(* CODESYS project IndraLogic.project

Project tree, tasks and I/O mapping:
  IndraMotionMlc1 : IndraMotion MLC L45, Bosch Rexroth AG, order no. R911170828, version 13.12.1.0
    application Application
      libraries: ML_TechInterface, 13.12.0.0 (System); RIL_LoopControl, 13.12.0.0 (System); ML_TechMotion, 13.12.3.0 (System); ML_TechRegi, 13.12.0.0 (System); RIL_ModbusTCP, 13.12.0.0 (System); RMB_TechWinder, 13.12.0.0 (System)
      task PlcTask (cyclic, interval 10 ms, priority 2) calls MAIN
      task MotionTask (externalevent, external event EVENT_OP_MODE_MOTION_CYCLIC, priority 1) calls MOTION
      AdjustPreset/
        program AdjustPreset [ST]
        program WriteExpectWindow [LD]
      global variables UserConstGlobal
      trace Trace (task MotionTask): 
      program MAIN [ST]
      Expectation Window Managment/
        ML_RegiCtrlExpectWinType01/
          function block ML_RegiCtrlExpectWinType01 [ST]: actShutdown
          DataTypes/
            data type ML_REGICTRL_EXPECTWIN_TYPE01
        ML_WriteExpectWinPosEdgeType01/
          Datatypes/
            data type ML_WRITE_EXPECT_WIN_TYPE01
          function block ML_WriteExpectWinPosEdgeType01 [ST]
      global variables UserVarGlobal
      ModbusComDataType/
        data type REGISTER_DATA
      STATE_MACHINE/
        program Machine [ST]
        program Winder [ST]
      program FormatC [ST]
      data type SETUP_STATE
      global variables MlcVarGlobal
      global variables GVL_MODBUS
      REF_SPEED/
        program SetVmaSpeed [ST]
      data type UTIL_STATE
      MAIN_PGM/
        program GravureState [ST]
        program ModbusCom [ST]
      program InsetterControl [LD]
      FLEXO_PGM/
        program TouchProbe [ST]
        program ProbeSetup [ST]
      Symbols
      INFEED/
      program MOTION [ST]
      AxisInterface/
        program _Readme [ST]
        function block TE_AxisInterface [ST]: actRetriggerOpMode, actPMSpecialErrors, mClearError, actPhaseShift, actAngleOffset, mGetOpMode, mSetOpMode, actSetupMode, actSyncAccVel, actCopyAxisData_HMI, mInitExtension
        Visualizations/
          ImcInterface/
            visualisation ImcStatus
            visualisation ImcControl
            visualisation ImcInterface_Status_Control
          SystemOverview/
            visualisation System_Overview_header
            visualisation System_Overview
            visualisation System_Overview_All_Axis
          AxisModes/
            visualisation Velocity_mode
            visualisation Position_mode
            visualisation Profile_mode
            visualisation Axis_Overview
            visualisation Synchronization_mode
          Utilities/
            visualisation PLC_load
            visualisation AdjustPosition
            visualisation AdjustVelocity
        function block TE_AxisInitAllAxisType01 [ST]
        function Version_AxisInterface_13V600 [ST]
        Documentation/
          program Visualisierungen [ST]
          program Visualisations [ST]
        program TE_AxisInterfaceType01Prog [ST]: actInitWarmStart
        Type/
          Status/
            data type TE_AXIS_DIAGNOSIS
            data type TE_AXIS_ADMIN_STATUS
            data type TE_AXIS_DATA_STATUS
            data type TE_AXIS_VEL_STATUS
            data type TE_AXIS_STATUS_TYPE01
            data type TE_AXIS_SETUP_MODE_STATUS
            data type TE_AXIS_POS_STATUS
            data type TE_AXIS_SYNC_STATUS
          Control/
            data type TE_AXIS_SETUP_MODE
            data type TE_AXIS_SYNCHRONISATION
            data type TE_AXIS_VELOCITY
            data type TE_AXIS_CONTROL_TYPE01
            data type TE_AXIS_POSITIONING
            data type TE_AXIS_ADMINISTRATION
          data type TE_PLC_CYCLES_TIME
        global variables Global_Axis_Interface
      program AUTO_REGISTER [ST]
      Utilities/
        program AllAxisHealthy [ST]
        program AllAxisAB [ST]
        program UnSynchronizePullroll [ST]
        function block FB_writevar [ST]
        program SynchronizePullroll [ST]
        program UnSynchronizeFlexo [ST]
        program InitAxis [ST]
        program SynchronizeFlexo [ST]
      REWIND/
        program WinderProcess [ST]
      data type STATE
      program POU [ST]
    Sercos_III_Master : SercosIII Master, Rexroth, order no. 1, version 13.2.2.0
    Inline_I_O : Inline I/O, Bosch Rexroth AG, version 12.8.2.0
    Not_Used : Not Used, Bosch Rexroth AG, version 12.2.0.0
    Not_Used_1 : Not Used, Bosch Rexroth AG, version 12.2.0.0
    Onboard_I_O : Onboard I/O, Bosch Rexroth AG, version 13.6.2.0
        input  x1 : BOOL  // OnboardIn.1.1
        input  x2 : BOOL  // OnboardIn.2.1
        input  x3 : BOOL  // OnboardIn.1.4
        input  x4 : BOOL  // OnboardIn.2.4
        input  x5 : BOOL  // OnboardIn.1.1
        input  x6 : BOOL  // OnboardIn.2.1
        input  x7 : BOOL  // OnboardIn.1.4
        input  x8 : BOOL  // OnboardIn.2.4
        unmapped channels: OnboardIn, OnboardOut
  text list GlobalTextList
*)

// IndraMotionMlc1/Application/AxisInterface/Type/Control/TE_AXIS_SETUP_MODE
TYPE TE_AXIS_SETUP_MODE :
  STRUCT
	  (* Enable setup mode  | Freigabe Einrichtbetrieb
      - activates Power                        | - aktiviert Antriebsfreigabe *)
    Enable:          BOOL;
 
	  (* Jog +            | Tippen +
        - activates ModeVelocity with pos. Vel   | - aktiviert ModeVelocity mit pos. Vel *)
    JogPlus:         BOOL;
 
	  (* Jog -            | Tippen -
       - activates ModeVelocity with pos. Vel   | - aktiviert ModeVelocity mit neg. Vel *)
    JogMinus:        BOOL;

	  (* Homing
      - activates ModeHoming|SetAbsRef|ModesPosAbs | activiert ModeHoming|SetAbsRef|ModesPosAbs
        depending on axistype/-configuration       | abhängig vom Achstyp/-konfiguration       *) 
    Homing: BOOL;
	
    Vel:    REAL:= 10; (* jog/homing velocity  | Tipp-/Referenzfahrgeschwindigkeit *)
	
    Accel:  REAL:= 10; (* jog/homing ac/deceleration  | Tipp/Referenzfahr (brems)beschleunigung *)
  END_STRUCT
END_TYPE

// IndraMotionMlc1/Application/AxisInterface/Type/Control/TE_AXIS_SYNCHRONISATION
    (*************** - setpoint of synchronous motion ******************)
TYPE TE_AXIS_SYNCHRONISATION EXTENDS MB_AXIS_SYNCHRONISATION:
STRUCT

    (* Electronic gear input revolution
      - "ModeSyncPhase", "ModeSyncVel", "ModeSyncCam", "ModeSyncProfile", "ModeFlexProfile"
      - RatioNumerator for MC_GearIn, MB_GearInPos, MC_CamIn, MB_MotionProfile, ML_FlexProfile 
      Note: cyclic checked AND transmitted on change (EnableCyclicScanning = TRUE) 
      ------------------------------------------------------------------------------
      Elektronisches Getriebe, Eingangsumdrehungen
      - "ModeSyncPhase", "ModeSyncVel", "ModeSyncCam", "ModeSyncProfile", "ModeFlexProfile"
      - RatioNumerator fuer MC_GearIn, MB_GearInPos, MC_CamIn, MB_MotionProfile, ML_FlexProfile 
      Hinweis: wird permanent zyklisch verarbeitet (EnableCyclicScanning = TRUE) *)
    // InputRevolution: UINT:=1;

    (* Electronic gear output revolution
      - "ModeSyncPhase", "ModeSyncVel", "ModeSyncCam", "ModeSyncProfile", "ModeFlexProfile"
      - RatioDenominator for MC_GearIn, MB_GearInPos, MC_CamIn, MB_MotionProfile, ML_FlexProfile 
      Note: cyclic checked AND transmitted on change (EnableCyclicScanning = TRUE)
      ------------------------------------------------------------------------------
      Elektronisches Getriebe, Ausgangsumdrehungen
      - "ModeSyncPhase", "ModeSyncVel", "ModeSyncCam", "ModeSyncProfile", "ModeFlexProfile"
      - RatioDenominator fuer MC_GearIn, MB_GearInPos, MC_CamIn, MB_MotionProfile, ML_FlexProfile 
      Hinweis: wird permanent zyklisch verarbeitet (EnableCyclicScanning = TRUE) *)
    // OutputRevolution: UINT:=1;

    (* Master fine adjust
      - "ModeSyncPhase", "ModeSyncVel", "ModeSyncCam", "ModeSyncProfile", "ModeFlexProfile"
      - MasterFineadjust for MC_GearIn, MB_GearInPos, MC_CamIn, MB_MotionProfile, ML_FlexProfile
      Note: cyclic checked AND transmitted on change (EnableCyclicScanning = TRUE) 
      ------------------------------------------------------------------------------
      Getriebe-Feinabgleich
      - "ModeSyncPhase", "ModeSyncVel", "ModeSyncCam", "ModeSyncProfile", "ModeFlexProfile"
      - MasterFineadjust fuer MC_GearIn, MB_GearInPos, MC_CamIn, MB_MotionProfile, ML_FlexProfile
      Hinweis: wird permanent zyklisch verarbeitet (EnableCyclicScanning = TRUE) *)
    // FineAdjust:    REAL:=0.0;

    (* Cam Shaft Distance
      - start moving with "ModeSyncCam"
      - CamShaftDist for MC_CamIn
      Note: cyclic checked AND transmitted on change (EnableCyclicScanning = TRUE) 
      ------------------------------------------------------------------------------
      Kurvenscheibe, Hub
      - Freigabe mit "ModeSyncCam" 
      - CamShaftDist fuer MC_CamIn
      Hinweis: wird permanent zyklisch verarbeitet (EnableCyclicScanning = TRUE) *)
    // CamShaftDistance: REAL:=360.0;

    (* Phase offset between master and slave axis
      - "ModeSyncPhase", "ModeSyncCam", "ModeSyncProfile", "ModeFlexProfile" 
      - PhaseShift for MB_PhasingSlave
      Note: cyclic checked AND transmitted on change (EnableCyclicScanning = TRUE) 
      ------------------------------------------------------------------------------
      Winkelversatz (Lagesollwert additiv)
      - "ModeSyncPhase", "ModeSyncCam", "ModeSyncProfile", "ModeFlexProfile" 
      - PhaseShift fuer MB_PhasingSlave
      Hinweis: wird permanent zyklisch verarbeitet (EnableCyclicScanning = TRUE) *)
    // PhaseOffset:   REAL:=0.0; 

    (* Velocity for the phase offset
      - "ModeSyncPhase", "ModeSyncCam", "ModeSyncProfile", "ModeFlexProfile"
      - Velocity for MB_PhasingSlave 
      ------------------------------------------------------------------------------
      Aufsynchronisier-Geschwindigkeit
      - "ModeSyncPhase", "ModeSyncCam", "ModeSyncProfile", "ModeFlexProfile"
      - Velocity fuer MB_PhasingSlave *)
	// PhaseOffsetVel: REAL:=1.0;

    (* Acceleration for the phase offset
      - "ModeSyncPhase", "ModeSyncCam", "ModeSyncProfile", "ModeFlexProfile" 
      - PhaseShift for MB_PhasingSlave
      ------------------------------------------------------------------------------
      Aufsynchronisier-Beschleunigung
      - Freigabe mit "ModeSyncPhase", "ModeSyncCam" oder "ModeSyncProfile"
      - PhaseShift fuer MB_PhasingSlave *)
    // PhaseOffsetAcc: REAL:=100.0;

    (* Synchronisation direction
      - values 'SHORTEST_WAY'; 'CATCH_UP' (always forward); 'SLOW_DOWN' (see RIL_CommonTypes.lib)
      - start moving with "ModeSyncPhase", "ModeSyncCam" or "ModeSyncProfile"
      - SyncMode for MB_GearInPos, MC_CamIn, MB_MotionProfile 
      ------------------------------------------------------------------------------
      Aufsynchronisier-Richtung
      - Werte 'SHORTEST_WAY'; 'CATCH_UP' (positiv); 'SLOW_DOWN' (siehe RIL_CommonTypes.lib)
      - Freigabe mit "ModeSyncPhase", "ModeSyncCam" oder "ModeSyncProfile"
      - SyncMode fuer MB_GearInPos, MC_CamIn, MB_MotionProfile *)
    // SyncDirection: MC_SYNC_DIRECTION:= SHORTEST_WAY;

    (* Start mode of the synchronisation
      - values 'ABSOLUTE'; 'RELATIVE' (see RIL_CommonTypes.lib)
      - start moving with "ModeSyncPhase", "ModeSyncCam" or "ModeSyncProfile"
      - StartMode for MB_GearInPos, MC_CamIn, MB_MotionProfile 
      ------------------------------------------------------------------------------
      Aufsynchronisier-Mode
      - Werte: 'ABSOLUTE'; 'RELATIVE' (siehe RIL_CommonTypes.lib)
      - Freigabe mit "ModeSyncPhase", "ModeSyncCam" oder "ModeSyncProfile"
      - StartMode fuer MB_GearInPos, MC_CamIn, MB_MotionProfile *)
    // StartMode:     MC_START_MODE:= ABSOLUTE;

    (* Number of the selected cam table
      - values 'CAM_TABLE_1'; 'CAM_TABLE_2' ... 'CAM_TABLE_8' (see RIL_CommonTypes.lib)
      - start moving with "ModeSyncCam" 
      - CamTableID for MC_CamIn
      Note: cyclic checked AND transmitted on change (EnableCyclicScanning = TRUE)
      ------------------------------------------------------------------------------
      Nummer Stuetzpunkt-Tabelle
      - Werte: 'CAM_TABLE_1'; 'CAM_TABLE_2' ... 'CAM_TABLE_8' (siehe RIL_CommonTypes.lib)
      - Freigabe mit "ModeSyncCam" 
      - CamTableID fuer MC_CamIn
      Hinweis: wird permanent zyklisch verarbeitet (EnableCyclicScanning = TRUE) *)
    // CamTableID:    MC_CAM_ID:= CAM_TABLE_1;

    (* -> AXIS_REF of the master axis
      - "ModeSyncPhase", "ModeSyncVel", "ModeSyncCam", "ModeSyncProfile", "ModeFlexProfile"
      - Master for MC_GearIn, MB_GearInPos, MC_CamIn, MB_MotionProfile, ML_FlexProfile 
      Note: cyclic checked AND transmitted on change (EnableCyclicScanning = TRUE)
      ------------------------------------------------------------------------------
      -> AXIS_REF der Leitachse
      - "ModeSyncPhase", "ModeSyncVel", "ModeSyncCam", "ModeSyncProfile", "ModeFlexProfile"
      - Master fuer MC_GearIn, MB_GearInPos, MC_CamIn, MB_MotionProfile, ML_FlexProfile 
         Hinweis: wird permanent zyklisch verarbeitet (EnableCyclicScanning = TRUE) *)
    // Master:    AXIS_REF    := (AxisNo := NO_OBJECT, CntrlNo := LOCAL_CNTRL);


    (*************** Extensions for profile operation modes *******************)
    (************* Erweiterungen für die Profil Betriebsarten *****************)
    (* Extensions for the operating modes MotionProfile and FlexProfile
       ------------------------------------------------------------------------------
       Erweiterungen füt die Betriebsarten MotionProfile und FlexProfile *)
    // Profile:     ML_AXIS_PROFILE;
	
  (* add your extensions below here, keep the elements above
     Erweiterungen hier einfuegen, Elemente oberhalb nicht veraendern *)

  (* user extensions | Anwender Erweiterungen *)

  // angle offset begin of profile | Winkelverschiebung Tabellenanfang
	AngleOffset:   REAL:= 0;  
	
  // Values for MB_Phasing | Werte für MB_Phasing
  // Additive master position command value
	PhaseShift:    REAL:=0.0;    
	PhaseShiftVel: REAL:=10.0;   // Additive master position velocity  
	PhaseShiftAcc: REAL:=100.0;  // Additive master position acceleration
		
  // A-0-2790 Synchronisation velocity | Aufsynchronisiergeschw.
  SyncVelocity:     REAL := 10.0; 

	// A-0-2791 Synchron. acceleration | Aufsynchronisierbeschleunigung
  SyncAcceleration: REAL := 10.0; 

END_STRUCT
END_TYPE

// IndraMotionMlc1/Application/AxisInterface/Type/Status/TE_AXIS_DIAGNOSIS
    (********** Diagnosis outputs - from motion control to logic control *****************)
    (********** Diagnose-Ausgaenge - Motion Control zur Logic Control    *****************)
TYPE TE_AXIS_DIAGNOSIS EXTENDS MB_AXIS_DIAGNOSIS:

STRUCT

  (* add your extensions below here |  Erweiterungen hier einfuegen*)

  (* user extensions | Anwender Erweiterungen *)


END_STRUCT

END_TYPE

// IndraMotionMlc1/Application/AxisInterface/Type/Control/TE_AXIS_VELOCITY
    (*************** - setpoints of velocity mode                    ************)
    (*************** - Sollwerte Geschwindigkeitsregelung (Freilauf) ************)
TYPE TE_AXIS_VELOCITY EXTENDS MB_AXIS_VELOCITY:
STRUCT

    (* Value of the maximum velocity (Unit: [u/s])
      - start moving with "ModeVel" (MC_MoveVelocity)
      Note: cyclic checked AND transmitted on change (EnableCyclicScanning = TRUE) 
      -----------------------------------------------------------------------------
      Geschwindigkeits-Sollwert, (Einheit: [u/s]) 
      - Freigabe mit "ModeVel" (MC_MoveVelocity)
      Hinweis: wird permanent zyklisch verarbeitet (EnableCyclicScanning = TRUE) *)
    // Velocity:        REAL:=0.0;

    (* Value of the acceleration and deceleration [u/s2] (always positive)
      - start moving with "ModeVel" (MC_MoveVelocity)
      -----------------------------------------------------------------------------
      Beschleunigung, (Einheit: [u/s2]) (immer positiv eingeben)            
      - Freigabe mit "ModeVel" (MC_MoveVelocity) *)
    // Acceleration:    REAL:=10.0;

    (* Value of the deceleration [u/s2] (always positive)
      - start moving with "ModeVel" (MC_MoveVelocity) 
      -----------------------------------------------------------------------------
      Verzoegerung, (Einheit: [u/s2]) (immer positiv eingeben)
      - Freigabe mit "ModeVel" (MC_MoveVelocity) *)
    // Deceleration:    REAL:=10.0;
	
(* add your extensions below here, keep the elements above
   Erweiterungen hier einfuegen, Elemente oberhalb nicht veraendern *)

(* user extensions | Anwender Erweiterungen *)

END_STRUCT
END_TYPE

// IndraMotionMlc1/Application/SETUP_STATE
TYPE SETUP_STATE :
(
	MECH_ACTIVE,MECH_UNSYNC,MECH_FORMAT_CH_P2,WRITE_NEW_GEARING,MECH_FORMAT_CH_P4,MECH_RESYNC,MECH_ERROR
);
END_TYPE

// IndraMotionMlc1/Application/AxisInterface/Type/Status/TE_AXIS_ADMIN_STATUS
    (********** Administrative outputs - from motion control to logic control *****************)
    (********** Administrative Ausgaenge - Motion Control zur Logic Control   *****************)
TYPE TE_AXIS_ADMIN_STATUS EXTENDS MB_AXIS_ADMIN_STATUS:

STRUCT
  (* add your extensions below here |  Erweiterungen hier einfuegen*)

  (* User extensions | Anwender Erweiterungen *)

 
END_STRUCT

END_TYPE

// IndraMotionMlc1/Application/AxisInterface/Type/Status/TE_AXIS_DATA_STATUS
TYPE TE_AXIS_DATA_STATUS :
STRUCT
	                  dwMotionProfileStatusBits_i     :DWORD;      (* A-0-2931 -RD- Motion profile status word *)
                      FlexProfil_Sync                 :BOOL;       (* A-0-3010.08 -RD- FlexProfile is in synchronisation *)
                      FlexProfil_Active               :BOOL;       (* A-0-3010.09 -RD- FlexProfile is active *)
                      FlexProfil_WaitForSwitching     :BOOL;       (* A-0-3010.10 -RD- FlexProfile is waiting for switching position *)
                      FlexProfil_Set0_Checked         :BOOL;       (* A-0-3010.16 -RD- FlexProfile Set0 is checked *)
                      FlexProfil_Set0_Ok              :BOOL;       (* A-0-3010.17 -RD- FlexProfile Set0 is ok *)
                      FlexProfil_Set1_Checked         :BOOL;       (* A-0-3010.18 -RD- FlexProfile Set0 is checked *)
                      FlexProfil_Set1_Ok              :BOOL;       (* A-0-3010.19 -RD- FlexProfile Set0 is ok *)
                      FlexProfil_Set2_Checked         :BOOL;       (* A-0-3010.20 -RD- FlexProfile Set0 is checked *)
                      FlexProfil_Set2_Ok              :BOOL;       (* A-0-3010.21 -RD- FlexProfile Set0 is ok *)
                      FlexProfil_Set3_Checked         :BOOL;       (* A-0-3010.22 -RD- FlexProfile Set0 is checked *)
                      FlexProfil_Set3_Ok              :BOOL;       (* A-0-3010.23 -RD- FlexProfile Set0 is ok *)
                      FlexProfil_EvtSet0_Checked      :BOOL;       (* A-0-3010.24 -RD- FlexProfile Event Set0 is checked *)
                      FlexProfil_EvtSet0_Ok           :BOOL;       (* A-0-3010.25 -RD- FlexProfile Event Set0 is ok *)
                      FlexProfil_EvtSet1_Checked      :BOOL;       (* A-0-3010.26 -RD- FlexProfile Event Set0 is checked *)
                      FlexProfil_EvtSet1_Ok           :BOOL;       (* A-0-3010.27 -RD- FlexProfile Event Set0 is ok *)
                      FlexProfil_EvtSet2_Checked      :BOOL;       (* A-0-3010.28 -RD- FlexProfile Event Set0 is checked *)
                      FlexProfil_EvtSet2_Ok           :BOOL;       (* A-0-3010.29 -RD- FlexProfile Event Set0 is ok *)
                      FlexProfil_EvtSet3_Checked      :BOOL;       (* A-0-3010.30 -RD- FlexProfile Event Set0 is checked *)
                      FlexProfil_EvtSet3_Ok           :BOOL;       (* A-0-3010.31 -RD- FlexProfile Event Set0 is ok *)
                      dwFlexProfileEventStatusBits_i  :DWORD;      (* A-0-3012 -RD- Condition status variable, FlexProfile *)

                      Axis_CamTab_0                   :BOOL;       (* A-0-0021.00 -RD- Cam shaft table BOOL 0 *)                
                      Axis_CamTab_1                   :BOOL;       (* A-0-0021.01 -RD- Cam shaft table BOOL 1 *)
                      Axis_CamTab_2                   :BOOL;       (* A-0-0021.02 -RD- Cam shaft table BOOL 2 (reserved) *)
                      Axis_CamSwitching               :BOOL;       (* A-0-0021.03 -RD- Status cam shaft distance switching *)
                      Axis_InVelocity                 :BOOL;       (* A-0-0021.04 -RD- Axis cmd velocity == actual velocity *)
                      Axis_Standstill                 :BOOL;       (* A-0-0021.05 -RD- Axis velocity <= A-0-0222 (standstill) *)
                      Axis_InPosition                 :BOOL;       (* A-0-0021.06 -RD- Axis cmd position == actual position *)
                      Axis_InSynchron                 :BOOL;       (* A-0-0021.07 -RD- Axis is in synchronisation *)
                      Axis_Warning                    :BOOL;       (* A-0-0021.08 -RD- Axis reports warning *)
                      Axis_Error                      :BOOL;       (* A-0-0021.09 -RD- Axis reports error *)
                      Axis_Homed                      :BOOL;       (* A-0-0021.10 -RD- Axis is relative / in homing *)
                      Axis_InTorque                   :BOOL;       (* A-0-0021.11 -RD- Axis cmd torque / force == actual torque *)
                      Axis_OperationMode              :BOOL;       (* A-0-0021.12 -RD- Axis is in operation mode (P4) *)
                      Axis_Inbb                       :BOOL;       (* A-0-0021.13 -RD- Axis is ready for power to the amplifier (bb) *)
                      Axis_InAb                       :BOOL;       (* A-0-0021.14 -RD- Axis is ready for power to the engine (Ab) *)
                      Axis_Power                      :BOOL;       (* A-0-0021.15 -RD- Axis has power on (AH_AF) *)
                      Axis_CmdActive                  :BOOL;       (* A-0-0021.16 -RD- Command active *)
                      Axis_ErrInProgress              :BOOL;       (* A-0-0021.17 -RD- Error reaction in progress *)
                      Axis_CyclicPosChannelOpen       :BOOL;       (* A-0-0021.18 -RD- Cyclic Position Channel is open for Axis *)          
                      Axis_InMasterPhaseOffset        :BOOL;       (* A-0-0021.19 -RD- Master Phase offset achieved *)
                      Axis_CyclicTrqChannelOpen       :BOOL;       (* A-0-0021.20 -RD- Cyclic Position Channel is open for Axis *)          
                      Axis_CyclicVelChannelOpen       :BOOL;       (* A-0-0021.21 -RD- Cyclic Position Channel is open for Axis *)          
                      Axis_CyclicAnaChannelOpen       :BOOL;       (* A-0-0021.22 -RD- Cyclic Position Channel is open for Axis *)          
                      ErrorStop                       :BOOL;       (* A-0-0022.00 -RD- Axis is in "ErrorStop" *)
                      Stopping                        :BOOL;       (* A-0-0022.01 -RD- Axis is in "Stopping" *)
                      Homing                          :BOOL;       (* A-0-0022.02 -RD- Command homing is active *)
                      PowerOn                         :BOOL;       (* A-0-0022.03 -RD- Axis got power *)
                      DiscreteMotion                  :BOOL;       (* A-0-0022.04 -RD- Axis is in "Discrete Motion" *)
                      ContinuousMotion                :BOOL;       (* A-0-0022.05 -RD- Axis is in "Continuous Motion" *)
                      SynchronizedMotion              :BOOL;       (* A-0-0022.06 -RD- Axis is in "Synchronized Motion" *)
                      Standstill                      :BOOL;       (* A-0-0022.07 -RD- Axis is stopped *)
                      CoordinatedMotion               :BOOL;       (* A-0-0022.08 -RD- Axis is in "CoordinatedMotion" *)
                      ControlledMotion                :BOOL;       (* A-0-0022.09 -RD- Axis is in "ControlledMotion" *)  
                      dwAxisCondition_i               :DWORD;      (* A-0-0024 -RD- Axis condition *)
                      rActualPosition_i               :REAL;       (* A-0-0100 -RD- Actual position *)
                      rActualVelocity_i               :REAL;       (* A-0-0102 -RD- Actual velocity *)
                      rActualTorqueForce_i            :REAL;       (* A-0-0110 -RD- Actual torque/force *)
                                                                                 
                    
                      wUserActualDataBitA_i           :WORD;      (* A-0-0562 -RD- User defined actual data BOOL number A, Type: WORD *)
                      wUserActualDataBitB_i           :WORD;      (* A-0-0565 -RD- User defined actual data BOOL number B, Type: WORD *)
                      wUserActualDataBitC_i           :WORD;      (* A-0-0568 -RD- User defined actual data BOOL number C, Type: WORD *)
                      wUserActualDataBitD_i           :WORD;      (* A-0-0571 -RD- User defined actual data BOOL number D, Type: WORD *)
                    
                      dwUserActualDataA_i             :SM_TYPES;  (* A-0-0521 -RD- Container user defined actual data A *)
                      dwUserActualDataB_i             :SM_TYPES;  (* A-0-0523 -RD- Container user defined actual data B *)
                      dwUserActualDataC_i             :SM_TYPES;  (* A-0-0525 -RD- Container user defined actual data C *)
                      dwUserActualDataD_i             :SM_TYPES;  (* A-0-0527 -RD- Container user defined actual data D *)
                      dwUserActualDataE_i             :SM_TYPES;  (* A-0-0529 -RD- Container user defined actual data E *)
                      dwUserActualDataF_i             :SM_TYPES;  (* A-0-0531 -RD- Container user defined actual data F *)
END_STRUCT
END_TYPE

// IndraMotionMlc1/Application/Expectation Window Managment/ML_WriteExpectWinPosEdgeType01/Datatypes/ML_WRITE_EXPECT_WIN_TYPE01
TYPE ML_WRITE_EXPECT_WIN_TYPE01 :
(
	STATE_IDLE,
	STATE_CHECK_VALIDITY,
	STATE_CALC_WINDOWS,
	STATE_WRITE_START_POS,
	STATE_WRITE_END_POS,
	STATE_ERROR,
	STATE_DONE,
	STATE_SHUTDOWN,
	STATE_RESET_PARAM_INST,
	STATE_DUMMY

);
END_TYPE

// IndraMotionMlc1/Application/AxisInterface/Type/Status/TE_AXIS_VEL_STATUS
    (********* Outputs of the following axis - from motion control to logic control **********)
    (********* Achs-Ausgaenge - Motion Control zur Logic Control                    **********)
TYPE TE_AXIS_VEL_STATUS  EXTENDS MB_AXIS_VEL_STATUS:
STRUCT
	(* -> outputs of the adjusting functionality for the velocity
      -> Ausgaenge fuer Tippbetrieb der Geschwindigkeit *)
    //Adjust: MB_AXIS_ADJUST_STATUS;
 
(* add your extensions below here, keep the elements above
   Erweiterungen hier einfuegen, Elemente oberhalb nicht veraendern *)

(* user extensions | Anwender Erweiterungen *)

END_STRUCT

END_TYPE

// IndraMotionMlc1/Application/AxisInterface/Type/Status/TE_AXIS_STATUS_TYPE01
    (********* Outputs of the following axis - from motion control to logic control **********)
TYPE TE_AXIS_STATUS_TYPE01:
  STRUCT
    (********* Outputs of the following axis - from motion control to logic control **********)

    PtrAxisData:  POINTER TO ML_AXISDATA_SM;
     (* Pointer to AxisData of this axis | Zeiger auf AxisData dieser Achse
      - Type .PtrAxisData^. for the intellisense menu | Eingabe .PtrAxisData^. fuer Auswahlmenue*)

    Admin:   TE_AXIS_ADMIN_STATUS; (* status of the axis | Achs-Status *)

    Diag:    TE_AXIS_DIAGNOSIS; (* axis diagnosis information, error, warning....
      Diagnose Informationen der Achse, Fehler, Warnung.... *)

    PosMode: TE_AXIS_POS_STATUS; (* Status operating mode positioning (absolute, rel. and add.)
      Statusmeldungen Positionierbetrieb (absolut, relativ und additiv) *)

    VelMode: TE_AXIS_VEL_STATUS; (* Status operating mode velocity control
      Statusmeldungen Geschwindigkeitsregelung (Freilauf) *)

    SyncMode: TE_AXIS_SYNC_STATUS; (* Status operating mode synchronisation (phase, vel, and cam)
      Statusmeldungen Synchronbetriebsarten (Winkelsync., Geschwindigkeitssync. und Kurvensch.)*)

    (* add your extensions below here, keep the elements above
       Erweiterungen hier einfuegen, Elemente oberhalb nicht veraendern *)
    (* user extensions | Anwender Erweiterungen *)
		(* Jog/Homing functionality | Tipp/Einrichtfunktionen *)
    SetupMode:  TE_AXIS_SETUP_MODE_STATUS;

    // AxisData for HMI (without data type "BIT")
	  AxisData_HMI:	TE_AXIS_DATA_STATUS;
	
  END_STRUCT
END_TYPE

// IndraMotionMlc1/Application/AxisInterface/Type/Status/TE_AXIS_SETUP_MODE_STATUS
TYPE TE_AXIS_SETUP_MODE_STATUS :
  STRUCT
	  (* Acknowledge setup mode  | Bestätigung Einrichtbetrieb
      - removed when _OpMode is oerwritten | - wird weggenommen, wenn _OpMode überschrieben wird *)
    EnableAck:   BOOL;
 
	  (* Acknowledge Homing 
      - ModeHoming|SetAbsRef|ModesPosAbs | ModeHoming|SetAbsRef|ModesPosAbs
        finished                         | abgeschlossen                    *) 
    HomingAck: 		BOOL;
	
  END_STRUCT
END_TYPE

// IndraMotionMlc1/Application/UTIL_STATE
TYPE UTIL_STATE :
(COMMAND,WAIT,DONE);
END_TYPE

// IndraMotionMlc1/Application/AxisInterface/Type/Control/TE_AXIS_CONTROL_TYPE01
TYPE TE_AXIS_CONTROL_TYPE01:

STRUCT
    Admin:      TE_AXIS_ADMINISTRATION; (* Administration of the axis | Verwaltung der Achse *)

    PosMode:    TE_AXIS_POSITIONING; (* operating mode positioning (absolute, rel. and additive)
      Positionierbetrieb (absolut, relativ und additiv) *)

    VelMode:    TE_AXIS_VELOCITY; (* operating mode velocity control | Geschwindigkeitsregelung *)

    SyncMode:   TE_AXIS_SYNCHRONISATION; (* operating mode synchronisation (phase, vel, and cam)
      Synchronbetriebsarten (Winkelsync., Geschwindigkeitssync. und Kurvenscheibe) *)

    (* add your extensions below here, keep the elements above
       Erweiterungen hier einfuegen, Elemente oberhalb nicht veraendern *)

    (* user extensions | Anwender Erweiterungen *)
    
	  // Jog/Homing functionality | Tipp/Einrichtfunktionen 
    SetupMode:  TE_AXIS_SETUP_MODE; 
	
END_STRUCT

END_TYPE

// IndraMotionMlc1/Application/ModbusComDataType/REGISTER_DATA
TYPE REGISTER_DATA :
STRUCT
	arWord:    ARRAY[0..20]OF WORD;     (* 1000 WORDS (%MB0000 - %MB999 ) *)
    (*arInt:     ARRAY[0..999]OF INT;      (* 1000 WORDS (%MB1000 - %MB1999) *)
	arUint:    ARRAY[0..999]OF UINT;     (* 1000 WORDS (%MB2000 - %MB2999) *)
	arDint:    ARRAY[0..499]OF DINT;     (* 1000 WORDS (%MB3000 - %MB3999) *)
	arUdint:   ARRAY[0..499]OF UDINT;    (* 1000 WORDS (%MB4000 - %MB4999) *)
	arReal:    ARRAY[0..499]OF REAL;     (* 1000 WORDS (%MB5000 - %MB5999) *)
	arString:  ARRAY[0..99]OF STRING(19);(* 1000 WORDS (%MB6000 - %MB6999) *)
	(* String(19): because 19 byte string + 1 byte end sign *)
	(* together 7000 WORDS *)*)
END_STRUCT
END_TYPE

// IndraMotionMlc1/Application/AxisInterface/Type/Status/TE_AXIS_POS_STATUS
    (********* Outputs of the following axis - from motion control to logic control **********)
    (********* Achs-Ausgaenge - Motion Control zur Logic Control                    **********)
TYPE TE_AXIS_POS_STATUS EXTENDS MB_AXIS_POS_STATUS:
STRUCT

	(* -> outputs of the adjusting functionality for the position
      -> Ausgaenge fuer Tippbetrieb der Position *)
    //Adjust: MB_AXIS_ADJUST_STATUS;
 
(* add your extensions below here, keep the elements above
   Erweiterungen hier einfuegen, Elemente oberhalb nicht veraendern *)

(* user extensions | Anwender Erweiterungen *)

END_STRUCT

END_TYPE

// IndraMotionMlc1/Application/AxisInterface/Type/Control/TE_AXIS_POSITIONING
    (*************** - setpoints of positioning mode ******************)
    (*************** - Positions-Sollwerte           ******************)
TYPE TE_AXIS_POSITIONING EXTENDS MB_AXIS_POSITIONING:
STRUCT

    (* position for an absolute move (in technical unit[u]) (negative or positive)
      - start moving with "ModePosAbs" (MC_MoveAbsolute)
      Note: cyclic checked AND transmitted on change (EnableCyclicScanning = TRUE) 
      ------------------------------------------------------------------------------
      Zielposition, absolut (Einheit: [u]) (negativ oder positiv)
      - Freigabe mit "ModePosAbs" (MC_MoveAbsolute)
      Hinweis: wird permanent zyklisch verarbeitet (EnableCyclicScanning = TRUE) *)
    // Position:        REAL;

    (* distance for a relative or additive move (in technical unit[u]) (negative or positive)
      - start moving with "ModePosRel" or "ModePosAdd" (MC_MoveRelative, MC_MoveAdditive) 
      Note: cyclic checked AND transmitted on change (EnableCyclicScanning = TRUE) 
      ------------------------------------------------------------------------------
      Relativer / additiver Sollwert (Einheit: [u]) (negativ oder positiv )
      - Freigabe mit "ModePosRel" oder "ModePosAdd" (MC_MoveRelative, MC_MoveAdditive) 
      Hinweis: wird permanent zyklisch verarbeitet (EnableCyclicScanning = TRUE) *)
     // Distance:        REAL;

    (* maximum velocity (always positive) (not necessarily reached) [u/s]
      - start moving with "ModePosAbs" or "ModePosRel" or "ModePosAdd" 
        (MC_MoveAbsolute, MC_MoveRelative, MC_MoveAdditive) 
      Note: cyclic checked AND transmitted on change (EnableCyclicScanning = TRUE) 
      ------------------------------------------------------------------------------
      Positioniergeschwindigkeit , (Einheit: [u/s]) (positiv eingeben)
      - Freigabe mit "ModePosAbs" oder "ModePosRel" oder "ModePosAdd" 
        (MC_MoveAbsolute, MC_MoveRelative, MC_MoveAdditive) 
      Hinweis: wird permanent zyklisch verarbeitet (EnableCyclicScanning = TRUE) *)
    // Velocity:        REAL:=10.0;

    (* Value of the acceleration (always positive) (increasing energy of the motor) [u/s2]
      - start moving with "ModePosAbs" or "ModePosRel" or "ModePosAdd" 
        (MC_MoveAbsolute, MC_MoveRelative, MC_MoveAdditive) 
      ------------------------------------------------------------------------------
      Beschleunigung (Einheit: [u/s2]) (nur positive Werte)             
      - Freigabe mit "ModePosAbs" oder "ModePosRel" oder "ModePosAdd" 
        (MC_MoveAbsolute, MC_MoveRelative, MC_MoveAdditive) *)
    // Acceleration:    REAL:=10.0;

    (* Value of the deceleration (always positive) (decreasing energy of the motor) [u/s2]
      - start moving with ModePosAbs or ModePosRel or ModePosAdd 
        (MC_MoveAbsolute, MC_MoveRelative, MC_MoveAdditive) 
      ------------------------------------------------------------------------------
      Verzoegerung, (Einheit: [u/s2]) (nur positive Werte)            
      - Freigabe mit "ModePosAbs" oder "ModePosRel" oder "ModePosAdd" 
        (MC_MoveAbsolute, MC_MoveRelative, MC_MoveAdditive) *)
    // Deceleration:    REAL:=10.0;
	
(* add your extensions below here, keep the elements above
   Erweiterungen hier einfuegen, Elemente oberhalb nicht veraendern *)

(* user extensions | Anwender Erweiterungen *)

END_STRUCT
END_TYPE

// IndraMotionMlc1/Application/AxisInterface/Type/Control/TE_AXIS_ADMINISTRATION
TYPE TE_AXIS_ADMINISTRATION EXTENDS MB_AXIS_ADMINISTRATION:
STRUCT
  (* add your extensions below here |  Erweiterungen hier einfuegen*)

  (* user extensions | Anwender Erweiterungen *)
  
  // Restart the same OpMode again, e.g. MoveRelative with same distance
  RetriggerOpMode: BOOL;	

END_STRUCT
END_TYPE

// IndraMotionMlc1/Application/AxisInterface/Type/Status/TE_AXIS_SYNC_STATUS
    (********* Outputs of the following axis - from motion control to logic control **********)
    (********* Achs-Ausgaenge - Motion Control zur Logic Control                    **********)
TYPE TE_AXIS_SYNC_STATUS EXTENDS MB_AXIS_SYNC_STATUS:
STRUCT
    // CamActiveID:      MC_CAM_ID; (* - ID of the active CamTable | - Nr. aktive Stuetzpunkt-Tab.*)

	(* - Number of the active motion profile set 0 or 1
      - Nummer des aktiven Satzes 0 oder 1 des Bewegungsprofils *)
    // ProfileActiveSet: UINT:= 0;  

	(* - Change of PhaseOffset is finished
      - Verstellung des PhaseOffset ist abgeschlossen  *)
    // PhasingSlaveDone: BOOL := FALSE; 

	(* adjusting | vertippen
      arAxisCntrl[].SyncMode.FineAdjust *)
    //AdjFineAdjust:       MB_AXIS_ADJUST_STATUS; 

	(* adjusting | vertippen
      arAxisCntrl[].SyncMode.CamShaftDistance *)
    //AdjCamShaftDistance: MB_AXIS_ADJUST_STATUS; 

	(* adjusting | vertippen
      arAxisCntrl[].SyncMode.PhaseOffset *)
    //AdjPhaseOffset:      MB_AXIS_ADJUST_STATUS;
	
  (* add your extensions below here, keep the elements above
     Erweiterungen hier einfuegen, Elemente oberhalb nicht veraendern *)

  (* user extensions | Anwender Erweiterungen *)
	// angle offset begin of profile | Winkelverschiebung Tabellenanfang 
  // transmission done | Übertragung abgeschlossen  
	AngleOffsetDone:   BOOL:= FALSE;   

  // Synchronisation velocity | Aufsynchronisiergeschw.
  // transmission done | Übertragung abgeschlossen  
  SyncVelocityDone:  BOOL:= FALSE;     

	// Synchron. acceleration | Aufsynchronisierbeschleunigung
  // transmission done | Übertragung abgeschlossen 
  SyncAccelerationDone: BOOL:= FALSE;  
	
  // Change of PhaseShift is finished | Verstellung des PhaseShift ist abgeschlossen 
  PhasingMasterDone: BOOL:=FALSE;
 
END_STRUCT

END_TYPE

// IndraMotionMlc1/Application/STATE

	
TYPE STATE :
(ERROR_CHECK,SETUP_PREPARE,SETUP_WAIT,SETUP_P2,SETUP_WRITEGEAR,SETUP_WRITEGEAR_WAIT,SETUP_P4,INIT_SYNC,INIT_VERIFY,
HOLD,RUN_PREPARE,RUN_DELAY,RUN,JOG_PREPARE,JOG_DELAY,JOG,JOG_WAIT,ERROR);


END_TYPE

// IndraMotionMlc1/Application/AxisInterface/Type/TE_PLC_CYCLES_TIME
TYPE TE_PLC_CYCLES_TIME :
STRUCT

     udiMinimumTime  : UDINT  := 1000000;
     udiActualTime   : UDINT  := 0;
     udiMaximumTime  : UDINT  := 0;

END_STRUCT
END_TYPE

// IndraMotionMlc1/Application/Expectation Window Managment/ML_RegiCtrlExpectWinType01/DataTypes/ML_REGICTRL_EXPECTWIN_TYPE01
TYPE ML_REGICTRL_EXPECTWIN_TYPE01 :
(
	
	STATE_IDLE,
	STATE_STORAGE_MODE_OFF,
	STATE_WAIT_REGI_IN_OPERATION,
	STATE_RESET_FB_INST,
	STATE_WAIT_REGI_SETPOINT_LOCK,
	STATE_RUN,
	STATE_SHUTDOWN,
	STATE_ERROR,
	STATE_DUMMY
);
END_TYPE

// IndraMotionMlc1/Application/UserConstGlobal
VAR_GLOBAL CONSTANT
  // define all possible axis, set to maximum axis index to preserve ressources 
  // set to a maximum of 32 for the L45 and 16? for the L25
  uiMAX_AXIS_INDEX:   UINT    := INT_TO_UINT(MB_MAX_AXIS_NUMBER);

  uiPRINT_AXIS_INDEX: UINT :=2;
END_VAR

// IndraMotionMlc1/Application/UserVarGlobal
VAR_GLOBAL 
  // Axis interface: command structure: define as RETAIN, to keep the values 
  // Note: on the L40.2 control, the RETAIN memory is slower then normal VAR, so define 
  //       this structure only as RETAIN when necessary 
  //  arAxisCtrl_gb: ARRAY [1..MAX_AXIS_NUM] OF MB_AXIS_CONTROL;
	
  // Axis interface: command structure 
  arAxisCtrl_gb: ARRAY [1..uiMAX_AXIS_INDEX] OF TE_AXIS_CONTROL_TYPE01;
	rExpectWindowPosEdgeStart_gb: REAL;
	rExpectWindowPosEdgeEnd_gb: REAL;
	rSetPointWindows_gb: REAL;
	Probe1Infeed: TOUCHPROBE_REF := (TouchProbeNo := TOUCHPROBE_DRIVE_1, CntrlNo := LOCAL_CNTRL);
END_VAR

VAR_GLOBAL
//----------------------------------- Machine status variables ----------------------------	

  // Axis interface: status structure 
  arAxisStatus_gb: ARRAY [1..uiMAX_AXIS_INDEX] OF TE_AXIS_STATUS_TYPE01;

  bRemoteOn_gb  : BOOL := TRUE;  // TRUE: Internal IL visu is active 
                                 // FALSE: PlcProg is active

								 	(*DEFINITION DU TOUCHPROB*)
tpDrv1: TOUCHPROBE_REF := (TouchProbeNo := TOUCHPROBE_DRIVE_1, CntrlNo := LOCAL_CNTRL);
  
END_VAR

// IndraMotionMlc1/Application/MlcVarGlobal
(* Automatically generated code by XLC/MLC. *)
(* Please don't edit, the code will be overwritten. For usercode use UserVarGlobal! *)
{attribute 'linkalways'}
VAR_GLOBAL CONSTANT

(*Real axis "Drive1" with axis number 1*)
Drive1: AXIS_REF :=(CntrlNo:=LOCAL_CNTRL,AxisNo:=AXIS_1);

(*Real axis "Drive2" with axis number 2*)
Drive2: AXIS_REF :=(CntrlNo:=LOCAL_CNTRL,AxisNo:=AXIS_2);

(*Real axis "Drive20" with axis number 20*)
Drive20: AXIS_REF :=(CntrlNo:=LOCAL_CNTRL,AxisNo:=AXIS_20);

(*Virtual axis "VMA_FT1" with axis number 30*)
VMA_FT1: AXIS_REF :=(CntrlNo:=LOCAL_CNTRL,AxisNo:=AXIS_30);


(*Probe 001*)
TouchProbe001: TOUCHPROBE_REF :=(CntrlNo:=LOCAL_CNTRL,TouchProbeNo:=TOUCHPROBE_1);

(*Probe 002*)
TouchProbe002: TOUCHPROBE_REF :=(CntrlNo:=LOCAL_CNTRL,TouchProbeNo:=TOUCHPROBE_2);

(*Probe 003*)
TouchProbe003: TOUCHPROBE_REF :=(CntrlNo:=LOCAL_CNTRL,TouchProbeNo:=TOUCHPROBE_3);

(*Probe 004*)
TouchProbe004: TOUCHPROBE_REF :=(CntrlNo:=LOCAL_CNTRL,TouchProbeNo:=TOUCHPROBE_4);

(*Probe 005*)
TouchProbe005: TOUCHPROBE_REF :=(CntrlNo:=LOCAL_CNTRL,TouchProbeNo:=TOUCHPROBE_5);

(*Probe 006*)
TouchProbe006: TOUCHPROBE_REF :=(CntrlNo:=LOCAL_CNTRL,TouchProbeNo:=TOUCHPROBE_6);

(*Probe 007*)
TouchProbe007: TOUCHPROBE_REF :=(CntrlNo:=LOCAL_CNTRL,TouchProbeNo:=TOUCHPROBE_7);

(*Probe 008*)
TouchProbe008: TOUCHPROBE_REF :=(CntrlNo:=LOCAL_CNTRL,TouchProbeNo:=TOUCHPROBE_8);

(*Probe 009*)
TouchProbe009: TOUCHPROBE_REF :=(CntrlNo:=LOCAL_CNTRL,TouchProbeNo:=TOUCHPROBE_9);

(*Probe 010*)
TouchProbe010: TOUCHPROBE_REF :=(CntrlNo:=LOCAL_CNTRL,TouchProbeNo:=TOUCHPROBE_10);

(*Probe 011*)
TouchProbe011: TOUCHPROBE_REF :=(CntrlNo:=LOCAL_CNTRL,TouchProbeNo:=TOUCHPROBE_11);

(*Probe 012*)
TouchProbe012: TOUCHPROBE_REF :=(CntrlNo:=LOCAL_CNTRL,TouchProbeNo:=TOUCHPROBE_12);

(*Probe 013*)
TouchProbe013: TOUCHPROBE_REF :=(CntrlNo:=LOCAL_CNTRL,TouchProbeNo:=TOUCHPROBE_13);

(*Probe 014*)
TouchProbe014: TOUCHPROBE_REF :=(CntrlNo:=LOCAL_CNTRL,TouchProbeNo:=TOUCHPROBE_14);

(*Probe 015*)
TouchProbe015: TOUCHPROBE_REF :=(CntrlNo:=LOCAL_CNTRL,TouchProbeNo:=TOUCHPROBE_15);

(*Probe 016*)
TouchProbe016: TOUCHPROBE_REF :=(CntrlNo:=LOCAL_CNTRL,TouchProbeNo:=TOUCHPROBE_16);

(*Probe 017*)
TouchProbe017: TOUCHPROBE_REF :=(CntrlNo:=LOCAL_CNTRL,TouchProbeNo:=TOUCHPROBE_17);

(*Probe 018*)
TouchProbe018: TOUCHPROBE_REF :=(CntrlNo:=LOCAL_CNTRL,TouchProbeNo:=TOUCHPROBE_18);

(*Probe 019*)
TouchProbe019: TOUCHPROBE_REF :=(CntrlNo:=LOCAL_CNTRL,TouchProbeNo:=TOUCHPROBE_19);

(*Probe 020*)
TouchProbe020: TOUCHPROBE_REF :=(CntrlNo:=LOCAL_CNTRL,TouchProbeNo:=TOUCHPROBE_20);

(*Probe 021*)
TouchProbe021: TOUCHPROBE_REF :=(CntrlNo:=LOCAL_CNTRL,TouchProbeNo:=TOUCHPROBE_21);

(*Probe 022*)
TouchProbe022: TOUCHPROBE_REF :=(CntrlNo:=LOCAL_CNTRL,TouchProbeNo:=TOUCHPROBE_22);

(*Probe 023*)
TouchProbe023: TOUCHPROBE_REF :=(CntrlNo:=LOCAL_CNTRL,TouchProbeNo:=TOUCHPROBE_23);

(*Probe 024*)
TouchProbe024: TOUCHPROBE_REF :=(CntrlNo:=LOCAL_CNTRL,TouchProbeNo:=TOUCHPROBE_24);

(*Probe 025*)
TouchProbe025: TOUCHPROBE_REF :=(CntrlNo:=LOCAL_CNTRL,TouchProbeNo:=TOUCHPROBE_25);

(*Probe 026*)
TouchProbe026: TOUCHPROBE_REF :=(CntrlNo:=LOCAL_CNTRL,TouchProbeNo:=TOUCHPROBE_26);

(*Probe 027*)
TouchProbe027: TOUCHPROBE_REF :=(CntrlNo:=LOCAL_CNTRL,TouchProbeNo:=TOUCHPROBE_27);

(*Probe 028*)
TouchProbe028: TOUCHPROBE_REF :=(CntrlNo:=LOCAL_CNTRL,TouchProbeNo:=TOUCHPROBE_28);

(*Probe 029*)
TouchProbe029: TOUCHPROBE_REF :=(CntrlNo:=LOCAL_CNTRL,TouchProbeNo:=TOUCHPROBE_29);

(*Probe 030*)
TouchProbe030: TOUCHPROBE_REF :=(CntrlNo:=LOCAL_CNTRL,TouchProbeNo:=TOUCHPROBE_30);

(*Probe 031*)
TouchProbe031: TOUCHPROBE_REF :=(CntrlNo:=LOCAL_CNTRL,TouchProbeNo:=TOUCHPROBE_31);

(*Probe 032*)
TouchProbe032: TOUCHPROBE_REF :=(CntrlNo:=LOCAL_CNTRL,TouchProbeNo:=TOUCHPROBE_32);

(*Probe 033*)
TouchProbe033: TOUCHPROBE_REF :=(CntrlNo:=LOCAL_CNTRL,TouchProbeNo:=TOUCHPROBE_33);

(*Probe 034*)
TouchProbe034: TOUCHPROBE_REF :=(CntrlNo:=LOCAL_CNTRL,TouchProbeNo:=TOUCHPROBE_34);

(*Probe 035*)
TouchProbe035: TOUCHPROBE_REF :=(CntrlNo:=LOCAL_CNTRL,TouchProbeNo:=TOUCHPROBE_35);

(*Probe 036*)
TouchProbe036: TOUCHPROBE_REF :=(CntrlNo:=LOCAL_CNTRL,TouchProbeNo:=TOUCHPROBE_36);

(*Probe 037*)
TouchProbe037: TOUCHPROBE_REF :=(CntrlNo:=LOCAL_CNTRL,TouchProbeNo:=TOUCHPROBE_37);

(*Probe 038*)
TouchProbe038: TOUCHPROBE_REF :=(CntrlNo:=LOCAL_CNTRL,TouchProbeNo:=TOUCHPROBE_38);

(*Probe 039*)
TouchProbe039: TOUCHPROBE_REF :=(CntrlNo:=LOCAL_CNTRL,TouchProbeNo:=TOUCHPROBE_39);

(*Probe 040*)
TouchProbe040: TOUCHPROBE_REF :=(CntrlNo:=LOCAL_CNTRL,TouchProbeNo:=TOUCHPROBE_40);

(*Probe 041*)
TouchProbe041: TOUCHPROBE_REF :=(CntrlNo:=LOCAL_CNTRL,TouchProbeNo:=TOUCHPROBE_41);

(*Probe 042*)
TouchProbe042: TOUCHPROBE_REF :=(CntrlNo:=LOCAL_CNTRL,TouchProbeNo:=TOUCHPROBE_42);

(*Probe 043*)
TouchProbe043: TOUCHPROBE_REF :=(CntrlNo:=LOCAL_CNTRL,TouchProbeNo:=TOUCHPROBE_43);

(*Probe 044*)
TouchProbe044: TOUCHPROBE_REF :=(CntrlNo:=LOCAL_CNTRL,TouchProbeNo:=TOUCHPROBE_44);

(*Probe 045*)
TouchProbe045: TOUCHPROBE_REF :=(CntrlNo:=LOCAL_CNTRL,TouchProbeNo:=TOUCHPROBE_45);

(*Probe 046*)
TouchProbe046: TOUCHPROBE_REF :=(CntrlNo:=LOCAL_CNTRL,TouchProbeNo:=TOUCHPROBE_46);

(*Probe 047*)
TouchProbe047: TOUCHPROBE_REF :=(CntrlNo:=LOCAL_CNTRL,TouchProbeNo:=TOUCHPROBE_47);

(*Probe 048*)
TouchProbe048: TOUCHPROBE_REF :=(CntrlNo:=LOCAL_CNTRL,TouchProbeNo:=TOUCHPROBE_48);

(*Probe 049*)
TouchProbe049: TOUCHPROBE_REF :=(CntrlNo:=LOCAL_CNTRL,TouchProbeNo:=TOUCHPROBE_49);

(*Probe 050*)
TouchProbe050: TOUCHPROBE_REF :=(CntrlNo:=LOCAL_CNTRL,TouchProbeNo:=TOUCHPROBE_50);

(*Probe 051*)
TouchProbe051: TOUCHPROBE_REF :=(CntrlNo:=LOCAL_CNTRL,TouchProbeNo:=TOUCHPROBE_51);

(*Probe 052*)
TouchProbe052: TOUCHPROBE_REF :=(CntrlNo:=LOCAL_CNTRL,TouchProbeNo:=TOUCHPROBE_52);

(*Probe 053*)
TouchProbe053: TOUCHPROBE_REF :=(CntrlNo:=LOCAL_CNTRL,TouchProbeNo:=TOUCHPROBE_53);

(*Probe 054*)
TouchProbe054: TOUCHPROBE_REF :=(CntrlNo:=LOCAL_CNTRL,TouchProbeNo:=TOUCHPROBE_54);

(*Probe 055*)
TouchProbe055: TOUCHPROBE_REF :=(CntrlNo:=LOCAL_CNTRL,TouchProbeNo:=TOUCHPROBE_55);

(*Probe 056*)
TouchProbe056: TOUCHPROBE_REF :=(CntrlNo:=LOCAL_CNTRL,TouchProbeNo:=TOUCHPROBE_56);

(*Probe 057*)
TouchProbe057: TOUCHPROBE_REF :=(CntrlNo:=LOCAL_CNTRL,TouchProbeNo:=TOUCHPROBE_57);

(*Probe 058*)
TouchProbe058: TOUCHPROBE_REF :=(CntrlNo:=LOCAL_CNTRL,TouchProbeNo:=TOUCHPROBE_58);

(*Probe 059*)
TouchProbe059: TOUCHPROBE_REF :=(CntrlNo:=LOCAL_CNTRL,TouchProbeNo:=TOUCHPROBE_59);

(*Probe 060*)
TouchProbe060: TOUCHPROBE_REF :=(CntrlNo:=LOCAL_CNTRL,TouchProbeNo:=TOUCHPROBE_60);

(*Probe 061*)
TouchProbe061: TOUCHPROBE_REF :=(CntrlNo:=LOCAL_CNTRL,TouchProbeNo:=TOUCHPROBE_61);

(*Probe 062*)
TouchProbe062: TOUCHPROBE_REF :=(CntrlNo:=LOCAL_CNTRL,TouchProbeNo:=TOUCHPROBE_62);

(*Probe 063*)
TouchProbe063: TOUCHPROBE_REF :=(CntrlNo:=LOCAL_CNTRL,TouchProbeNo:=TOUCHPROBE_63);

(*Probe 064*)
TouchProbe064: TOUCHPROBE_REF :=(CntrlNo:=LOCAL_CNTRL,TouchProbeNo:=TOUCHPROBE_64);

(*Probe 065*)
TouchProbe065: TOUCHPROBE_REF :=(CntrlNo:=LOCAL_CNTRL,TouchProbeNo:=TOUCHPROBE_65);

(*Probe 066*)
TouchProbe066: TOUCHPROBE_REF :=(CntrlNo:=LOCAL_CNTRL,TouchProbeNo:=TOUCHPROBE_66);

(*Probe 067*)
TouchProbe067: TOUCHPROBE_REF :=(CntrlNo:=LOCAL_CNTRL,TouchProbeNo:=TOUCHPROBE_67);

(*Probe 068*)
TouchProbe068: TOUCHPROBE_REF :=(CntrlNo:=LOCAL_CNTRL,TouchProbeNo:=TOUCHPROBE_68);

(*Probe 069*)
TouchProbe069: TOUCHPROBE_REF :=(CntrlNo:=LOCAL_CNTRL,TouchProbeNo:=TOUCHPROBE_69);

(*Probe 070*)
TouchProbe070: TOUCHPROBE_REF :=(CntrlNo:=LOCAL_CNTRL,TouchProbeNo:=TOUCHPROBE_70);

(*Probe 071*)
TouchProbe071: TOUCHPROBE_REF :=(CntrlNo:=LOCAL_CNTRL,TouchProbeNo:=TOUCHPROBE_71);

(*Probe 072*)
TouchProbe072: TOUCHPROBE_REF :=(CntrlNo:=LOCAL_CNTRL,TouchProbeNo:=TOUCHPROBE_72);

(*Probe 073*)
TouchProbe073: TOUCHPROBE_REF :=(CntrlNo:=LOCAL_CNTRL,TouchProbeNo:=TOUCHPROBE_73);

(*Probe 074*)
TouchProbe074: TOUCHPROBE_REF :=(CntrlNo:=LOCAL_CNTRL,TouchProbeNo:=TOUCHPROBE_74);

(*Probe 075*)
TouchProbe075: TOUCHPROBE_REF :=(CntrlNo:=LOCAL_CNTRL,TouchProbeNo:=TOUCHPROBE_75);

(*Probe 076*)
TouchProbe076: TOUCHPROBE_REF :=(CntrlNo:=LOCAL_CNTRL,TouchProbeNo:=TOUCHPROBE_76);

(*Probe 077*)
TouchProbe077: TOUCHPROBE_REF :=(CntrlNo:=LOCAL_CNTRL,TouchProbeNo:=TOUCHPROBE_77);

(*Probe 078*)
TouchProbe078: TOUCHPROBE_REF :=(CntrlNo:=LOCAL_CNTRL,TouchProbeNo:=TOUCHPROBE_78);

(*Probe 079*)
TouchProbe079: TOUCHPROBE_REF :=(CntrlNo:=LOCAL_CNTRL,TouchProbeNo:=TOUCHPROBE_79);

(*Probe 080*)
TouchProbe080: TOUCHPROBE_REF :=(CntrlNo:=LOCAL_CNTRL,TouchProbeNo:=TOUCHPROBE_80);

(*Probe 081*)
TouchProbe081: TOUCHPROBE_REF :=(CntrlNo:=LOCAL_CNTRL,TouchProbeNo:=TOUCHPROBE_81);

(*Probe 082*)
TouchProbe082: TOUCHPROBE_REF :=(CntrlNo:=LOCAL_CNTRL,TouchProbeNo:=TOUCHPROBE_82);

(*Probe 083*)
TouchProbe083: TOUCHPROBE_REF :=(CntrlNo:=LOCAL_CNTRL,TouchProbeNo:=TOUCHPROBE_83);

(*Probe 084*)
TouchProbe084: TOUCHPROBE_REF :=(CntrlNo:=LOCAL_CNTRL,TouchProbeNo:=TOUCHPROBE_84);

(*Probe 085*)
TouchProbe085: TOUCHPROBE_REF :=(CntrlNo:=LOCAL_CNTRL,TouchProbeNo:=TOUCHPROBE_85);

(*Probe 086*)
TouchProbe086: TOUCHPROBE_REF :=(CntrlNo:=LOCAL_CNTRL,TouchProbeNo:=TOUCHPROBE_86);

(*Probe 087*)
TouchProbe087: TOUCHPROBE_REF :=(CntrlNo:=LOCAL_CNTRL,TouchProbeNo:=TOUCHPROBE_87);

(*Probe 088*)
TouchProbe088: TOUCHPROBE_REF :=(CntrlNo:=LOCAL_CNTRL,TouchProbeNo:=TOUCHPROBE_88);

(*Probe 089*)
TouchProbe089: TOUCHPROBE_REF :=(CntrlNo:=LOCAL_CNTRL,TouchProbeNo:=TOUCHPROBE_89);

(*Probe 090*)
TouchProbe090: TOUCHPROBE_REF :=(CntrlNo:=LOCAL_CNTRL,TouchProbeNo:=TOUCHPROBE_90);

(*Probe 091*)
TouchProbe091: TOUCHPROBE_REF :=(CntrlNo:=LOCAL_CNTRL,TouchProbeNo:=TOUCHPROBE_91);

(*Probe 092*)
TouchProbe092: TOUCHPROBE_REF :=(CntrlNo:=LOCAL_CNTRL,TouchProbeNo:=TOUCHPROBE_92);

(*Probe 093*)
TouchProbe093: TOUCHPROBE_REF :=(CntrlNo:=LOCAL_CNTRL,TouchProbeNo:=TOUCHPROBE_93);

(*Probe 094*)
TouchProbe094: TOUCHPROBE_REF :=(CntrlNo:=LOCAL_CNTRL,TouchProbeNo:=TOUCHPROBE_94);

(*Probe 095*)
TouchProbe095: TOUCHPROBE_REF :=(CntrlNo:=LOCAL_CNTRL,TouchProbeNo:=TOUCHPROBE_95);

(*Probe 096*)
TouchProbe096: TOUCHPROBE_REF :=(CntrlNo:=LOCAL_CNTRL,TouchProbeNo:=TOUCHPROBE_96);

(*Probe 097*)
TouchProbe097: TOUCHPROBE_REF :=(CntrlNo:=LOCAL_CNTRL,TouchProbeNo:=TOUCHPROBE_97);

(*Probe 098*)
TouchProbe098: TOUCHPROBE_REF :=(CntrlNo:=LOCAL_CNTRL,TouchProbeNo:=TOUCHPROBE_98);

(*Probe 099*)
TouchProbe099: TOUCHPROBE_REF :=(CntrlNo:=LOCAL_CNTRL,TouchProbeNo:=TOUCHPROBE_99);

(*Probe 100*)
TouchProbe100: TOUCHPROBE_REF :=(CntrlNo:=LOCAL_CNTRL,TouchProbeNo:=TOUCHPROBE_100);

END_VAR

// IndraMotionMlc1/Application/GVL_MODBUS
VAR_GLOBAL
	

	//RegisterData:          REGISTER_DATA;              (* Holding Register data area for FC3, FC6, FC16 and FC23        *)
	bGratuve_Tens_Inc_ETH_i	:BOOL;
	bGratuve_Tens_Dec_ETH_i	:BOOL;
	bGravure_Reg_Adv_ETH_q	:BOOL;
	bGravure_Reg_Ret_ETH_q	:BOOL;
	bGravureOn_ETH_q		:BOOL;
	
	bRegAdvance_ETH_i		:BOOL;
	bRegRetard_ETH_i		:BOOL;
	bGravure_Jog_Adv_HMI_i	:BOOL;
	bGravure_Jog_Ret_HMI_i	:BOOL;
	
	bInfeedOn_ETH_q			:BOOL;
	bInfeedManual_ETH_q		:BOOL;
	bInfeed_Inc_Tens_HMI_i	:BOOL;
	bInfeed_Dec_Tens_HMI_i	:BOOL;
	
	uiGearingRatio_HMI_q	:BOOL;
	
	bGravure_StatusError_HMI_q		:BOOL;
	bGravure_StatusSynch_HMI_q		:BOOL;
	bGravure_StatusSlowRot_HMI_q	:BOOL;
	bGravure_StatusDisabled_HMI_q	:BOOL;
	
	bInfeed_StatusError_HMI_q		:BOOL;
	bInfeed_StatusSynch_HMI_q		:BOOL;
	bInfeed_StatusSlowRot_HMI_q		:BOOL;
	bInfeed_StatusDisabled_HMI_q	:BOOL;
	
	bGravure_ResetDrive_HMI_i:BOOL;
	bInfeed_ResetDrive_HMI_i:BOOL;
	bRewindPID_Out_i:BOOL;
	bGravureSlowRot_ETH_i:BOOL;
	
	
		bGravureFB:BOOL:= TRUE;
		bGravureRegiOn_HMI_i:	BOOL;
		bInfeedRegiOn_HMI_i:	BOOL;
		bGravureNipActive_i:	BOOL;
		bPauseRegiOn_HMI_i: BOOL;
		bSetPtLckRegiCtrl_HMI_i: BOOL;
		bSetPtLckRegiCtrlAck_HMI_q: BOOL;
		bTouchProbeInOp_HMI_q:BOOL;
		uiDetectedPosEdge_gb:UINT;
		rCurrentValue_HMI_q:REAL;
		rRegiCtrlSetPoint: REAL;
		rDeviation_gb:REAL;
	
		rDeviationMil_gb:REAL;
		rSetPointWindowsMil_gb:REAL;
		
		
		
	dwDeviation_gb:DWORD;
	dwDeviation_low_gb:DWORD;
	dwDeviation_high_gb:DWORD;


	dwRegiCtrlSetPoint_gb:DWORD;
	dwRegiCtrlSetPoint_low_gb:DWORD;
	dwRegiCtrlSetPoint_high_gb:DWORD;
	dwLoadcellTension_gb:DWORD;
	
	dwRegAdjustLow_gb:DWORD;
	dwRegAdjustHigh_gb:DWORD;
	dwRegAdjust_gb:DWORD;
	
	arDrive: ARRAY[1..2] OF AXIS_REF;
	arProbe: ARRAY[1..2] OF TOUCHPROBE_REF;
END_VAR

// IndraMotionMlc1/Application/AxisInterface/Global_Axis_Interface
{attribute 'linkalways'}
VAR_GLOBAL
    (* Axis number for the visualization screens *)
    VisuAxisNo : INT := 1;
END_VAR

// IndraMotionMlc1/Application/MAIN
PROGRAM MAIN
VAR
	
ii:UINT;
bBogus:BOOL;
uiState1:UTIL_STATE;
uiState2:UTIL_STATE;
bRun_HMI_i:BOOL;
bJog_HMI_i:BOOL;
bStop_HMI_i:BOOL;
bReset_HMI_i:BOOL;
bOkToRun_i:BOOL:=TRUE;
bOkToJog_i:BOOL:=TRUE;
bFault_i:BOOL;
bInterlock_i:BOOL:=TRUE;
bSetup_HMI_i:BOOL;
newSTATE:STATE;
bSetupDone_i:BOOL;

	arFlexoAxis:	ARRAY[1..20] OF AXIS_REF;
	arPullrollAxis: ARRAY[1..20] OF AXIS_REF;
	arWindingAxis:	ARRAY[1..20] OF AXIS_REF;
	
	index:UINT;
		
	arFlexoPointer: POINTER TO ARRAY[1..20] OF AXIS_REF;
	test:AXIS_REF;
	uiAxisTotNumNew: UINT;
	
	
	bUnsync:BOOL;
	bSync:BOOL;
	binit:BOOL:=FALSE;	
	bAllAxisAB:BOOL;
	bAllFlexoSync:BOOL;
	bAllFlexoUnsync: BOOL;
	
	fbRunButton: R_TRIG;
	fbSetupButton: R_TRIG;
	
	rRepeat_i	:REAL	:= 1.0;
	iFormat_i	:INT := 4800;	//8 inches format
	rRunSpd		:REAL:= 100.0;
	rJogSpd		:REAL:= 10.0;
	bWriteExec: BOOL;
	
	bRewIntrlock:BOOL;
END_VAR


VAR CONSTANT
	uiNUM_FLEXO		: UINT:=2;
	uiNUM_PULLROLL	: UINT:=0;
	uiNUM_WINDER	: UINT:=1;
	iTeethConstant	: INT :=8;
END_VAR

IF TE_AxisInterfaceType01Prog.InitDone=FALSE THEN
	RETURN;
END_IF

//AXIS DEFINITION
arFlexoAxis[1] := arAxisCtrl_gb[Drive1.AxisNo].Admin.Axis;
arFlexoAxis[2] := arAxisCtrl_gb[Drive2.AxisNo].Admin.Axis;
//Winders
arWindingAxis[1]:= arAxisCtrl_gb[Drive20.AxisNo].Admin.Axis;

IF NOT binit THEN InitAxis(arAxisPointer:=ADR(arFlexoAxis) , uiNUM_FLEXO_F:= uiNUM_FLEXO);
				  InitAxis(arAxisPointer:=ADR(arWindingAxis) , uiNUM_FLEXO_F:= uiNUM_WINDER);

ELSE	//______    INIT IS OVER       ______!!!!!!!



bReset_HMI_i;
//THIS FUNCTION IS THE CORE OF THE MACHINE POSSIBLE STATES
Winder(
	arAxisPointer:= ADR(arWindingAxis), 
	uiNUM_FLEXO_F:= uiNUM_WINDER, 
	MACHINE_STATE_i:= newSTATE, 
	iGearValue:= 1, 
	bRewIntrlock=> bRewIntrlock);


Machine(
	arAxisPointer_M	:=ADR(arFlexoAxis),
	uiNUM_FLEXO_M	:=uiNUM_FLEXO,
	bRun_i			:=	bRun_HMI_i , 
	bJog_i			:=	bJog_HMI_i , 
	bStop_i			:=	bStop_HMI_i , 
	okToRun			:=	bOkToRun_i , 
	okToJog			:=	bOkToJog_i , 
	bFault			:=	bFault_i, 
	bIntrlock		:=	bInterlock_i, 
	bSetup_i		:=	 bSetup_HMI_i,
	bWriteExec		:=  bWriteExec, 
	CURRENT_STATE_OUT=> newSTATE );	

rRepeat_i:=INT_TO_REAL(iFormat_i/iTeethConstant)/ 100.0;

//THIS FUNCTION SETS SPEED ACCORDING TO THE FORMAT 
SetVmaSpeed(
	arAxisPointer:=ADR(arFlexoAxis) , 
	uiNUM_FLEXO_F:=uiNUM_FLEXO , 
	rFormat:=rRepeat_i , 
	rRunSpeedDemandFPM:=rRunSpd , 
	rJogSpeedDemandFPM:= rJogSpd, 
	uiState:=newSTATE , 
	);
//SET FORMAT
//THIS FUNCTION SETS MECHANICAL GEAR DEPENDING ON THE PLATE CYLINDER USED
//IT ALSO ADJUSTS THE SYNC_REVOLUTION TO COMPENSATES THE ADJUSTMENT OF VMA SPEED
FormatC(
	arAxisPointer:= ADR(arFlexoAxis), 
	uiNUM_FLEXO_F:= uiNUM_FLEXO , 
	MACHINE_STATE_i:= newSTATE , 
	iGearValue:=     iFormat_i , 
	bExecute:= bWriteExec , 
	bSetupDone_i=> );	

//GravureState();
//InfeedState();
ModbusCom();
//POU();

END_IF
binit:= TRUE;

END_PROGRAM

// IndraMotionMlc1/Application/AxisInterface/TE_AxisInterfaceType01Prog
PROGRAM TE_AxisInterfaceType01Prog
(*#############################################################################################
  #############################################################################################  

   General Header   
  ---------------------------------------------------------------------------------------------  
   Shortdescription       : Cyclic execution of the Axis-Interface (POS, VEL and SYNC mode)
   Version                : see Version_GAT_compact_11V200 
   Name                   : DCC/EAM3 (KG)
   Date                   : see Version_GAT_compact_11V200
   Company                : see Version_GAT_compact_11V200
   Target                 : see Version_GAT_compact_11V200
   Functional description : This program executes cyclic the axis interface FB for all axes.
                            The execution time of the axis interface FB is measured.
   Handling specials      : The global arrays of the axis-interface must be named arAxisCtrl[]
                            and arAxisStatus[]
  ---------------------------------------------------------------------------------------------  
    
   Additional Header   
  ---------------------------------------------------------------------------------------------  
  #############################################################################################  
  #############################################################################################*)
(*
                                     ******************
                                     *   DISCLAIMER   *
                                     ******************
   It is acknowledged that with regard to these software programs and program modules free of
   charge, Bosch Rexroth's usually practised, in-house test and release procedures have not 
   been accomplished. These software programs and program modules free of charge serve only as
   an example for possible applications.  They are intended as a help in order to obtain addi-
   tional experience regarding function, operation, performance and capacity of a maybe later 
   issued series release. Therefore Bosch Rexroth disclaims any liability and rejects to assume
   responsibility that these software programs or program modules, including any information 
   and data stored in those programs, are suitable for any intended use or that these programs
   will work without errors in any combination with the data processing environment. Providing
   you with these software programs shall neither constitute a claim for technical support nor
   for any other remedy for defects. Any claims for damages of any nature and for any legal
   reason arising from installing or using these software programs or program modules are ex-
   cluded, unless these damages was caused by Bosch Rexroth`s statutory representatives or em-
   ployees by wilful misconduct or by gross negligence or liability is compulsory in accordance
   with the German product liability law. In any case Bosch Rexroth`s liability for any conse-
   quential or incidental damages such as, but not limited to loss of profit, loss of pro-
   duction or loss of data is excluded.      
*)
(*---------------------------------------------------------------------------------------------*)
VAR_INPUT
  ClearError: BOOL;		// clear internal errors of the program
END_VAR
VAR_OUTPUT
  InitDone: BOOL;		// Init is done, AxisInterface is ready to operate
  Error: BOOL;			// internal error of the program
  ErrorID: ERROR_CODE;
  ErrorIdent: ERROR_STRUCT;
END_VAR
VAR CONSTANT
   STATE_FIRST_INIT       : UINT := 0;
   STATE_WAIT_FOR_PHASE2  : UINT := 1;
   STATE_INIT_P2          : UINT := 2;
   STATE_WAIT_FOR_PHASE4  : UINT := 3;
   STATE_INIT_P4          : UINT := 4;
   STATE_WAIT_FOR_NOT_P4  : UINT := 5;
   STATE_PRG_ERROR        : UINT := 9;
   
   dwADD1_STATE_MACHINE_ERROR: DWORD := 16#00000006;
   dwADD2_STATE_MACHINE_ERROR: DWORD := 16#00000000;
   
END_VAR
VAR
    fbAxisInitAllAxis: TE_AxisInitAllAxisType01; //  basic init of arAxisCtrl structure 

    uiState                 : UINT := STATE_FIRST_INIT; // statemachine
	  // Flag that the inputs of the FB are set
	  bInitReferencesDone: BOOL; 
  
    fbAxis                    : ARRAY [1..uiMAX_AXIS_INDEX] OF TE_AxisInterface;
	  uiLoop                    : UINT := 1;
	  // time measurement
    udiStartTime              : UDINT;
    udiStopTime               : UDINT;
	  udiActCycleTime           : UDINT;
    stCyclesTime              : TE_PLC_CYCLES_TIME;
END_VAR

// -------------------------------------------------------------------------------- 
// state-machine: do the warmstart initialisation everytime we reach SERCOS phase 4 
// -------------------------------------------------------------------------------- 
CASE uiState OF

  STATE_FIRST_INIT:
    // ---------------------------------------------------------------------------------
    // Step: Done only once when PLC program starts.           
    // ---------------------------------------------------------------------------------
   	FOR uiLoop := 1 TO uiMAX_AXIS_INDEX DO
		 	fbAxis[uiLoop].mInitExtension(uiLoop);
		END_FOR
		bInitReferencesDone := TRUE; // Inputs are set, FB can be called	
    uiState := STATE_WAIT_FOR_PHASE2;
  
  STATE_WAIT_FOR_PHASE2:
    // --------------------------------------------------------------------------------- 
    // Step: Wait for SERCOS phase P2;                                                   
    // Done cyclic when we are in phases < 2                                             
    // --------------------------------------------------------------------------------- 
    IF (ImcStatus.Admin.ModeStatus_P2 = TRUE) THEN
      uiState := STATE_INIT_P2;
      InitDone := FALSE;      
		ELSIF( (ImcStatus.Admin.PwrUpModeAck = TRUE) AND (ImcStatus.Admin._OpModeAck > IMC_MODE_STATUS_P2) ) THEN
  	// E.g. PL program download in P4, go directly to P4
      uiState := STATE_WAIT_FOR_PHASE4;
      InitDone := FALSE;      
    END_IF
	
  STATE_INIT_P2:
    // --------------------------------------------------------------------------------- 
    // Step: Action actInitWarmStart. Done when reaching parameter mode.                 
    // --------------------------------------------------------------------------------- 
    actInitWarmStart();

  STATE_WAIT_FOR_PHASE4:
    // --------------------------------------------------------------------------------- 
    // Step: Wait for SERCOS phase P4;                                                   
    // Done cyclic when we are not in phase 4                                            
    // --------------------------------------------------------------------------------- 
    IF( ImcStatus.Admin.ModeStatus_P3 = TRUE ) THEN
      InitDone := FALSE; // reset the InitDone so with reaching bb it is already TRUE       
    ELSIF( ImcStatus.Admin.ModeStatus_BB = TRUE )THEN
      uiState := STATE_INIT_P4;
      InitDone := FALSE;      
    END_IF


  STATE_INIT_P4:
    // --------------------------------------------------------------------------------- 
    // Step: Action actInitWarmStart. Done when reaching operating mode.                 
    // --------------------------------------------------------------------------------- 
    actInitWarmStart();


  STATE_WAIT_FOR_NOT_P4:
    // --------------------------------------------------------------------------------- 
    // Step: Check SECROS phase changes from P4                                          
    // Done cyclic when we are in phase 4                                                
	// Set bAxisInterfaceInitDone to FALSE to enforce a re-init, e.g. changing A-0-0024  
    // --------------------------------------------------------------------------------- 

    // Check if we have left phase 4 
    IF( (ImcStatus.Admin.ModeStatus_BB = FALSE) OR (InitDone = FALSE) ) THEN
      // We have left phase 4 -> re-init the axis interface 
      uiState := STATE_WAIT_FOR_PHASE4;
    END_IF
	
  STATE_PRG_ERROR:
    IF ClearError = TRUE THEN
      // clear error information
      Error := FALSE;
  InitDone := FALSE; // enforce a new init 
      uiState := STATE_WAIT_FOR_PHASE4;
    END_IF
	
  ELSE
	// -------------------------------------------- 
    // DEFAULT case -> Signal error !!!                      
    // -------------------------------------------- 
    Error := TRUE;
    // set error information
    ErrorID := STATE_MACHINE_ERROR;
    ErrorIdent.Table := F_RELATED_TABLE;
	ErrorIdent.Additional1 := dwADD1_STATE_MACHINE_ERROR;
	ErrorIdent.Additional2 := dwADD2_STATE_MACHINE_ERROR;
    uiState := STATE_PRG_ERROR; 

END_CASE

udiStartTime := IL_HighResTimeTick(TRUE); // latch starting time 

IF (InitDone AND bInitReferencesDone) THEN
  FOR uiLoop := 1 TO uiMAX_AXIS_INDEX DO
    fbAxis[uiLoop]( ); // call FB, inputs are already set....
  END_FOR
END_IF  

udiStopTime := IL_HighResTimeTick(TRUE); // latch end time 

// calculate actual runtime and store MIN and MAX 
udiActCycleTime := IL_HighResTimeDiff(udiStartTime,udiStopTime);

stCyclesTime.udiActualTime := udiActCycleTime;

IF (stCyclesTime.udiMaximumTime < udiActCycleTime) THEN
  stCyclesTime.udiMaximumTime := udiActCycleTime;
END_IF

IF (stCyclesTime.udiMinimumTime > udiActCycleTime) THEN
  stCyclestime.udiMinimumTime := udiActCycleTime;
END_IF

ACTION actInitWarmStart:
// --------------------------------------------------------------------------------- 
// Action actInitWarmStart: Done when reaching parameter mode (P2)                   
// and again when reaching operating mode (phase 4)             	             
// --------------------------------------------------------------------------------- 

// ############################################ 
// Step: Basic Init of arAxisCtrl_gb for all axes  
// ############################################ 
fbAxisInitAllAxis(
  Execute:= TRUE,
  ReadModuloValue:=TRUE,
  EnableCyclicScanning:=TRUE );

IF(fbAxisInitAllAxis.Error = TRUE) THEN
  // -------------------------------------------- 
  // Signal error !!!                      
  // -------------------------------------------- 
  Error := TRUE;
  // copy error information
  ErrorID := fbAxisInitAllAxis.ErrorID;
  ErrorIdent := fbAxisInitAllAxis.ErrorIdent;
  // reset FB 
  fbAxisinitAllAxis( Execute := FALSE );
  // go to error state
  uiState := STATE_PRG_ERROR; 
  
ELSIF(fbAxisInitAllAxis.Done = TRUE) THEN
  // basic init of control structure
  // example: virtual axis 2 follows virtual axis 1
 // arAxisCtrl_gb[MyVirtualAxis2.AxisNo].SyncMode.Master := MyVirtualAxis1;

  // -------------------------------------------- 
  // Signal init is finished                      
  // -------------------------------------------- 
  InitDone := TRUE; // Init is finished 
  // reset FB 
  fbAxisinitAllAxis( Execute := FALSE );
  

  // ---------------------------------------------------------------------------------
  // End of this state by increasing uiState (call from STATE_INIT_P2 or STATE_INIT_P4)                                          
  // ---------------------------------------------------------------------------------
  uiState := uiState + 1;
END_IF
END_ACTION

END_PROGRAM

// IndraMotionMlc1/Application/STATE_MACHINE/Machine
PROGRAM Machine
VAR
	

	//(HOLD,RUN_PREPARE,RUN_DELAY,RUN,JOG_PREPARE,JOG_DELAY,JOG,JOG_WAIT);
	bRunHold_out:BOOL;
	ENABLE	:BOOL;
	CONDITION1:BOOL;
	CONDITION2:BOOL;
	SUCCEED:BOOL;
	CURRENT_STATE : STATE; 
	fbRunHold		: R_TRIG;
	fbRunPrepare		: R_TRIG;
	

	
	bRunActive:BOOL;
	fbPrepareTimer: TON ;
	bPrepareTimer:BOOL;
	
	fbJogRtrig1: R_TRIG;
	fbJogFtrig1: F_TRIG;
	fbSetupRtrig1: R_TRIG;
	bAllAxisSynch: BOOL;
	bSync: BOOL := TRUE;
	bUnSync:BOOL := TRUE;
	bAllFlexoSync: BOOL;
	bAllFlexoUnsync: BOOL;
	uiState1: UTIL_STATE;
	uiState2: UTIL_STATE;

	bGoodtogo:BOOL;
	bAllAxisHealthy:BOOL;
	fbNew: TON;
	bTimerOn: BOOL;
END_VAR

VAR_INPUT
	
arAxisPointer_M: POINTER TO ARRAY[1..20] OF AXIS_REF;
uiNUM_FLEXO_M: UINT;
bRun_i:BOOL;
bJog_i:BOOL;
bStop_i:BOOL;	
okToRun:BOOL;
okToJog:BOOL;
bFault		:BOOL;	//Fault = true means no go
bIntrlock	:BOOL;	//Interlock = false means no go
bSetup_i:BOOL;


END_VAR
VAR_IN_OUT
	bWriteExec:BOOL;
END_VAR

VAR_OUTPUT
	CURRENT_STATE_OUT:STATE;
	
END_VAR


CURRENT_STATE_OUT := CURRENT_STATE;
fbRunHold(CLK:=bRun_i , Q=>bRunHold_out );
fbPrepareTimer(IN:=bPrepareTimer , PT:=T#5.0S , Q=> , ET=> );


fbJogRtrig1(CLK:=bJog_i , Q=> );
fbJogFtrig1(CLK:=bJog_i , Q=> );
fbSetupRtrig1(CLK:=bSetup_i , Q=> );

fbNew(IN:=bTimerOn , PT:= T#10S, Q=> , ET=> );
		
				 

CASE CURRENT_STATE OF 

	ERROR_CHECK:
	//CHECK IF ANY ERROR EXISTS
		AllAxisHealthy(arAxisPointer:=arAxisPointer_M , uiNUM_FLEXO_F:=uiNUM_FLEXO_M , bAllAxisHealthy=>bAllAxisHealthy );
		IF NOT bAllAxisHealthy THEN
			ImcCtrl.Admin.ClearError := TRUE;
		ELSE
			ImcCtrl.Admin.ClearError := FALSE;
		END_IF
		
		IF bAllAxisHealthy THEN
			CURRENT_STATE := SETUP_PREPARE;
		END_IF
	SETUP_PREPARE:
	
	//UNSYNC THE FLEXO DRIVES
		ImcCtrl.Admin.ClearError := FALSE;
		bUnSync := TRUE;
		UnSynchronizeFlexo(arAxisPointer:=arAxisPointer_M , uiNUM_FLEXO_F:=uiNUM_FLEXO_M , bExecute:=bUnSync , 
				bAllAxisAB=>  bAllFlexoUnsync, uiState=>uiState2 );
		
		arAxisCtrl_gb[VMA_FT1.AxisNo].Admin._OpMode.en:=ModeAB;		
		
		IF NOT bUnSync AND arAxisStatus_gb[VMA_FT1.AxisNo].Admin._OpModeAck=ModeAB THEN
			
			CURRENT_STATE := SETUP_P2;
		END_IF	
		
	SETUP_WAIT:
		
		bTimerOn:= TRUE;
		IF fbNew.Q THEN
			bTimerOn:= FALSE;
			CURRENT_STATE := SETUP_P2;
		END_IF	
	SETUP_P2:
		ImcCtrl.Admin._OpMode:=(IMC_MODE_CTRL_P2);
		IF ImcStatus.Admin._OpModeAck=IMC_MODE_CTRL_P2 THEN
				CURRENT_STATE := SETUP_WRITEGEAR;
		END_IF
		bPrepareTimer:= TRUE;//start timer
		//IF fbPrepareTimer.Q THEN
			//	CURRENT_STATE := ERROR;
		//END_IF

	SETUP_WRITEGEAR:
		ImcCtrl.Admin.ClearError := TRUE;
		bWriteExec := TRUE;
		CURRENT_STATE := SETUP_WRITEGEAR_WAIT;
	
	SETUP_WRITEGEAR_WAIT:	
		
		IF NOT bWriteExec THEN
			CURRENT_STATE := SETUP_P4;
		END_IF
	SETUP_P4:
		ImcCtrl.Admin.ClearError := TRUE;
		ImcCtrl.Admin._OpMode:=IMC_MODE_CTRL_BB;
		IF ImcStatus.Admin._OpModeAck=IMC_MODE_STATUS_BB THEN
			CURRENT_STATE := INIT_SYNC;
		END_IF
	
	INIT_SYNC:	//SYNCH ALL AXIS
		ImcCtrl.Admin.ClearError := TRUE;
		bSync:=TRUE;
		SynchronizeFlexo(arAxisPointer:=arAxisPointer_M , uiNUM_FLEXO_F:=uiNUM_FLEXO_M , bExecute:=bSync ,
				 bAllFlexoSync=> bAllFlexoSync,uiState=>uiState1);
	
		
		IF uiState1=DONE THEN
			CURRENT_STATE := HOLD;
		END_IF
	INIT_VERIFY:	//VERIFY SYNCH ALL AXIS
		
	HOLD: 
		//IN HOLD ALL AXIS ARE SYNC TO VMA	
		bPrepareTimer:= FALSE;
		IF  fbRunHold.Q=TRUE AND okToRun AND (NOT bFault) AND bIntrlock AND NOT bStop_i THEN
			CURRENT_STATE := RUN_PREPARE;
		ELSIF  fbJogRtrig1.Q=TRUE AND okToJog AND (NOT bFault) AND bIntrlock AND NOT bStop_i THEN
			CURRENT_STATE := JOG;
		ELSIF  fbSetupRtrig1.Q=TRUE THEN
			CURRENT_STATE := SETUP_PREPARE;
		END_IF
		
	
		
	
	RUN_PREPARE:
		IF  fbRunHold.Q=TRUE AND okToRun AND (NOT bFault) AND bIntrlock AND NOT bStop_i THEN
			CURRENT_STATE := RUN_DELAY;
		END_IF
		
		
	RUN_DELAY: 
		bPrepareTimer:= TRUE;
		IF  fbPrepareTimer.Q THEN
			CURRENT_STATE := RUN;
		END_IF
		
	RUN: 
		
		bRunActive := TRUE;
		
		//arAxisCtrl_gb[VMA_FT1].Admin._OpMode.b.MODE_VEL
		arAxisCtrl_gb[VMA_FT1.AxisNo].Admin._OpMode.en := ModeVel;
		
	

		IF  bJog_i=TRUE AND okToJog AND (NOT bFault) AND bIntrlock AND NOT bStop_i THEN
			CURRENT_STATE := JOG;
		END_IF
		
		
		IF (NOT okToRun) OR  bFault OR (NOT bIntrlock) OR bStop_i THEN
			CURRENT_STATE := HOLD;
		END_IF
		
	JOG:
		
		IF fbJogFtrig1.Q AND bRunActive=TRUE AND okToRun AND (NOT bFault) AND bIntrlock AND NOT bStop_i THEN
			CURRENT_STATE := RUN;
		END_IF

		IF   (fbJogFtrig1.Q AND (NOT bRunActive)) OR (NOT okToJog) OR bFault OR (NOT bIntrlock) OR bStop_i THEN
			CURRENT_STATE := HOLD;
		END_IF
	
	JOG_WAIT:
			CURRENT_STATE := HOLD;

	ERROR:
		;
END_CASE;

END_PROGRAM

// IndraMotionMlc1/Application/Utilities/AllAxisHealthy
PROGRAM AllAxisHealthy
VAR_INPUT
	arAxisPointer: POINTER TO ARRAY[1..20] OF AXIS_REF;
	uiNUM_FLEXO_F: UINT;
END_VAR
VAR_OUTPUT
	
	bAllAxisHealthy:BOOL;
END_VAR
VAR
	index : UINT :=1;
END_VAR

bAllAxisHealthy := TRUE;

FOR index:=1 TO uiNUM_FLEXO_F BY 1 DO
	IF 	arAxisStatus_gb[arAxisPointer^[index].AxisNo].Diag.Error THEN
		
		bAllAxisHealthy := FALSE;
	ELSE
		;
	END_IF
END_FOR

IF ImcStatus.Diag.Error THEN
	bAllAxisHealthy := FALSE;
END_IF

END_PROGRAM

// IndraMotionMlc1/Application/Utilities/UnSynchronizeFlexo
PROGRAM UnSynchronizeFlexo
VAR_INPUT
	
	arAxisPointer: POINTER TO ARRAY[1..20] OF AXIS_REF;
	uiNUM_FLEXO_F: UINT;
	
END_VAR
VAR_OUTPUT
	bAllAxisAB : BOOL;
	uiState:UTIL_STATE;
END_VAR
VAR
	index : UINT;
	fbExec: R_TRIG;
END_VAR
VAR_IN_OUT
	bExecute:BOOL;
END_VAR

CASE uiState OF 

	COMMAND:
		IF bExecute THEN
			FOR index:=1 TO uiNUM_FLEXO_F BY 1 DO	
					arAxisCtrl_gb[arAxisPointer^[index].AxisNo].Admin._OpMode.en:=ModeAB;
					uiState := WAIT;
			END_FOR
		
		END_IF
		
	WAIT:
		bAllAxisAB := TRUE;
		FOR index:=1 TO uiNUM_FLEXO_F BY 1 DO	
				IF 	arAxisStatus_gb[arAxisPointer^[index].AxisNo].Admin._OpModeAck=ModeAB THEN
				;//do nothing (it stays true)
				ELSE
					bAllAxisAB := FALSE;
				END_IF
		END_FOR
		IF bAllAxisAB THEN
			uiState := DONE;
		END_IF
	DONE:
		
			bExecute := FALSE;
			uiState := COMMAND;
		
END_CASE;

END_PROGRAM

// IndraMotionMlc1/Application/Utilities/SynchronizeFlexo
PROGRAM SynchronizeFlexo
VAR_INPUT
	
	arAxisPointer: POINTER TO ARRAY[1..20] OF AXIS_REF;
	uiNUM_FLEXO_F: UINT;
	
END_VAR
VAR_OUTPUT
	bAllFlexoSync : BOOL;
	uiState:UTIL_STATE;
END_VAR
VAR
	index : UINT :=1;
	
	fbExec: R_TRIG;
	
	cnt:UINT:=0;
END_VAR
VAR_IN_OUT
	bExecute:BOOL;
	
END_VAR

cnt := cnt + 1 ;
CASE uiState OF 

	COMMAND:
		IF bExecute THEN
			FOR index:=1 TO uiNUM_FLEXO_F BY 1 DO	
					arAxisCtrl_gb[arAxisPointer^[index].AxisNo].Admin._OpMode.en:=ModeSyncPhase;
			END_FOR
			//arAxisCtrl_gb[arAxisPointer^[index].AxisNo].Admin._OpMode.en:=ModeSyncPhase;
			uiState := WAIT;
		END_IF
		
	WAIT:
		bAllFlexoSync := TRUE;
		FOR index:=1 TO uiNUM_FLEXO_F BY 1 DO	
				IF 	arAxisStatus_gb[arAxisPointer^[index].AxisNo].Admin._OpModeAck=ModeSyncPhase THEN
					;//do nothing (it stays true)
				ELSE
					bAllFlexoSync := FALSE;
				END_IF
		END_FOR
	
		IF bAllFlexoSync THEN
			uiState := DONE;
		
		END_IF
	DONE:
		
			bExecute := FALSE;
			uiState := COMMAND;
		
END_CASE;

END_PROGRAM

// IndraMotionMlc1/Application/AxisInterface/TE_AxisInitAllAxisType01
(* Initialisation of the Axis-Interface (POS, VEL and SYNC mode)
  #############################################################################################
  #############################################################################################  

   General Header   
  ---------------------------------------------------------------------------------------------  
   Shortdescription       : Initialisation of the Axis-Interface (POS, VEL and SYNC mode)
   Version                : 1.01  
   Name                   : BRC/EAM3 (KG,PoVa)
   Date                   : 2008-May-05  
   Company                : Bosch Rexroth Electric Drives and Controls GmbH  
   Target                 : IndraMotion MLC   
   Functional description : This functionblocks initialises the data structures for the
                            axis interface. All available axes (C-0-0484) are activated.
   Handling specials      : The global arrays of the axis-interface must be named arAxisCtrl_gb[]
                            and arAxisStatus_gb[]
  ---------------------------------------------------------------------------------------------  
    
   Additional Header   
     The following structure elements are set by this function block:
      arAxisCtrl_gb[].Admin._OpMode.en = ModeAB
      arAxisCtrl_gb[].Admin.ClearError = FALSE      
      arAxisCtrl_gb[].Admin.LockInputChanges = FALSE       
      arAxisCtrl_gb[].Admin.SetAbsRef = FALSE      
      arAxisCtrl_gb[].Admin.Axis.CntrlNo = LOCAL_CNTRL;
      arAxisCtrl_gb[].Admin.Axis.AxisNo = AXIS_1 .. AXIS_n
      arAxisCtrl_gb[].PosMode.Adjust.Enable = FALSE       
      arAxisCtrl_gb[].VelMode.Adjust.Enable = FALSE       
      arAxisCtrl_gb[].SyncMode.AdjCamShaftDist.Enable = FALSE       
      arAxisCtrl_gb[].SyncMode.AdjFineadjust.Enable = FALSE         
      arAxisCtrl_gb[].SyncMode.AdjPhaseOffset.Enable = FALSE        
      arAxisCtrl_gb[].Comment = A-0-0002

      arAxisStatus_gb[].Active = TRUE for active axis ( C-0-0484 )
      arAxisStatus_gb[].Admin.AxisFeatures = type set with value of A-0-0004 for all axis

    Only when ReadModuloValue = TRUE and the axis is rotatoric:
      arAxisCtrl_gb[iAxisNo].PosMode.Adjust.ModuloValue = A-0-0045
      arAxisCtrl_gb[iAxisNo].SyncMode.AdjPhaseOffset.ModuloValue = A-0-045
      arAxisCtrl_gb[iAxisNo].VelMode.Adjust.ModuloValue = 0
      arAxisCtrl_gb[iAxisNo].SyncMode.AdjCamShaftDist.ModuloValue = 0
      arAxisCtrl_gb[iAxisNo].SyncMode.AdjFineadjust.ModuloValue = 0

  ---------------------------------------------------------------------------------------------  
     
     
     
  ---------------------------------------------------------------------------------------------  

  #############################################################################################  
  #############################################################################################*)
(*
                                     ******************
                                     *   DISCLAIMER   *
                                     ******************
   It is acknowledged that with regard to these software programs and program modules free of
   charge, Bosch Rexroth's usually practised, in-house test and release procedures have not 
   been accomplished. These software programs and program modules free of charge serve only as
   an example for possible applications.  They are intended as a help in order to obtain addi-
   tional experience regarding function, operation, performance and capacity of a maybe later 
   issued series release. Therefore Bosch Rexroth disclaims any liability and rejects to assume
   responsibility that these software programs or program modules, including any information 
   and data stored in those programs, are suitable for any intended use or that these programs
   will work without errors in any combination with the data processing environment. Providing
   you with these software programs shall neither constitute a claim for technical support nor
   for any other remedy for defects. Any claims for damages of any nature and for any legal
   reason arising from installing or using these software programs or program modules are ex-
   cluded, unless these damages was caused by Bosch Rexroth`s statutory representatives or em-
   ployees by wilful misconduct or by gross negligence or liability is compulsory in accordance
   with the German product liability law. In any case Bosch Rexroth`s liability for any conse-
   quential or incidental damages such as, but not limited to loss of profit, loss of pro-
   duction or loss of data is excluded.      
*)
(*---------------------------------------------------------------------------------------------*)

FUNCTION_BLOCK TE_AxisInitAllAxisType01

VAR_INPUT
    Execute         : BOOL;            (* start execution with rising edge *)
    ReadModuloValue : BOOL := TRUE;    (* Read parameters A59 and A45 and write the modulo value
                                          for rotatoric axis to the adjustment structure of PosMode
                                          SyncMode.AdjPhaseOffset and set modulo value to 0 for all
                                          other adjusted values. Activate before "Execute" *)
    EnableCyclicScanning : BOOL := TRUE; (* Enable the cyclic check and transmission of changed
                                            inputs for the actual operating mode
                                            - relevant for the values in AxisCtrl with 
                                              "Note: cyclic checked AND transmitted on change" *)
END_VAR

VAR_OUTPUT
    Done        : BOOL := FALSE;       (* Is SET when FB has finished operation *)
    Active      : BOOL := FALSE;       (* Is SET when FB is active (not in idle mode) *)
    Error       : BOOL := FALSE;       (* ErrorFlag *)
    ErrorID     : ERROR_CODE;          (* Error identification, Errorcode *)
    ErrorIdent  : ERROR_STRUCT;        (* Error identification *)
END_VAR

VAR
    bOldExecute         : BOOL := FALSE;
    uiState             : UINT := 0;
    stDummyAxis         : AXIS_REF;
    arBuffer            : ARRAY [1..(uiMAX_AXIS_INDEX*2)] OF INT;
    fbReadListParaC484  : MB_ReadListParameter;
    uiAxisNo            : UINT   := 1;
    Axis                : AXIS_REF;
    fbAxisInitType01    : MB_AxisInitType01;
END_VAR

VAR CONSTANT
   STATE_DO_NOTHING             : UINT := 0;
   STATE_READ_C484              : UINT := 1;
   STATE_CHK_AXIS               : UINT := 2;
   STATE_START_INIT             : UINT := 3;
END_VAR

(* Detect rising edge *)
IF( (Execute = TRUE) AND (bOldExecute = FALSE) ) THEN
     uistate := STATE_READ_C484;
END_IF

CASE uiState OF

    STATE_DO_NOTHING:
      IF( Execute = FALSE ) THEN
        (* RESET everything *)
        Done    := FALSE;
        Active  := FALSE;
        Error   := FALSE;
        uiAxisNo := 1;
      END_IF;

    STATE_READ_C484:
      (* ############################################### *)
      (* Step: Read C-0-0484 "Axes configuration list"   *)
      (* ############################################### *)

      fbReadListParaC484(
        Execute           := TRUE,
        ParameterNumber   := FP_C_0_0484,
        NoOfBytes         := (uiMAX_AXIS_INDEX*4),
        ValueAdr          := ADR(arBuffer),
        Axis              := stDummyAxis);

      IF ( fbReadListParaC484.Done = TRUE ) THEN
        (* reset FB *)
        fbReadListParaC484(
          Execute    := FALSE,
          Axis       := stDummyAxis);
        uiState := STATE_CHK_AXIS;
        uiAxisNo := 1;
      END_IF

  STATE_CHK_AXIS:
    (* ############################################ *)
    (* Step: Check all configured axis              *)
    (* ############################################ *)
    IF ( uiAxisNo <= uiMAX_AXIS_INDEX ) THEN
      (* activate, when axis type not equal 0 *)
      IF ( arBuffer[2*uiAxisNo - 1] <> 0 ) THEN
        uiState      := STATE_START_INIT;
        Axis.AxisNo  := uiAxisNo;
        Axis.CntrlNo := LOCAL_CNTRL;
      ELSE
        uiAxisNo := uiAxisNo + 1;
      END_IF

    ELSE
      Done    := TRUE;
      Active  := FALSE;
      uiState := STATE_DO_NOTHING;
    END_IF

  STATE_START_INIT:
    (* ############################################ *)
    (* Step: Initialize all configured axis         *)
    (* ############################################ *)

    (* call FB ML_AxisInitType01 -> initialize the axis *)
    fbAxisInitType01(
      Execute              := TRUE,
      ReadModuloValue      := ReadModuloValue,
      EnableCyclicScanning := EnableCyclicScanning,
      AdminCtrl            := arAxisCtrl_gb[uiAxisNo].Admin,
      PosModeCtrl          := arAxisCtrl_gb[uiAxisNo].PosMode,
      VelModeCtrl          := arAxisCtrl_gb[uiAxisNo].VelMode,
      SyncModeCtrl         := arAxisCtrl_gb[uiAxisNo].SyncMode,
      AxisDataPtrStatus    := arAxisStatus_gb[uiAxisNo].PtrAxisData,
      AdminStatus          := arAxisStatus_gb[uiAxisNo].Admin,
      DiagStatus           := arAxisStatus_gb[uiAxisNo].Diag,
      Axis                 := Axis);
    IF ( fbAxisInitType01.Error = TRUE ) THEN
      Error      := fbAxisInitType01.Error;
      ErrorID    := fbAxisInitType01.ErrorID;
      ErrorIdent := fbAxisInitType01.ErrorIdent;
    END_IF

    IF ( fbAxisInitType01.Done = TRUE ) THEN
      (* restart ML_AxisInitType01 *)
      fbAxisInitType01(
        Execute            := FALSE,
        AdminCtrl          := arAxisCtrl_gb[uiAxisNo].Admin,
        PosModeCtrl        := arAxisCtrl_gb[uiAxisNo].PosMode,
        VelModeCtrl        := arAxisCtrl_gb[uiAxisNo].VelMode,
        SyncModeCtrl       := arAxisCtrl_gb[uiAxisNo].SyncMode,
        AxisDataPtrStatus  := arAxisStatus_gb[uiAxisNo].PtrAxisData,
        AdminStatus        := arAxisStatus_gb[uiAxisNo].Admin,
        DiagStatus         := arAxisStatus_gb[uiAxisNo].Diag,
        Axis               := Axis);
      (* check next axis *)
      uiAxisNo := uiAxisNo + 1;
      (* proceed with STATE_DO -> check next configured axis *)
      uiState := STATE_CHK_AXIS;

    END_IF

END_CASE

(* Edge detection *)
bOldExecute := Execute;

END_FUNCTION_BLOCK

// IndraMotionMlc1/Application/AxisInterface/TE_AxisInterface
FUNCTION_BLOCK TE_AxisInterface EXTENDS MB_AxisInterfaceType01
(*#############################################################################################
  #############################################################################################  

  General Header   
  ---------------------------------------------------------------------------------------------  
  Shortdescription       : AxisInterface Example 
  Version                : see Version_AxisInterface_xxVyyy
  Name                   : DCC/EAM (DT/KG)
  Date                   : see Version_AxisInterface_xxVyyy
  Company                : see Version_AxisInterface_xxVyyy
  Target                 : see Version_AxisInterface_xxVyyy
  Functional description : Location in order to extend the AxisInterface functionality
  Handling specials      : This functionality is automatically assigned to the task the approriate
                           axis is assigned to
  ---------------------------------------------------------------------------------------------  
  
  Additional Header   
  ---------------------------------------------------------------------------------------------  

  ---------------------------------------------------------------------------------------------  

###############################################################################################  
###############################################################################################*)
(*
                                     ******************
                                     *   DISCLAIMER   *
                                     ******************
   It is acknowledged that with regard to these software programs and program modules free of
   charge, Bosch Rexroth's usually practised, in-house test and release procedures have not 
   been accomplished. These software programs and program modules free of charge serve only as
   an example for possible applications.  They are intended as a help in order to obtain addi-
   tional experience regarding function, operation, performance and capacity of a maybe later 
   issued series release. Therefore Bosch Rexroth disclaims any liability and rejects to assume
   responsibility that these software programs or program modules, including any information 
   and data stored in those programs, are suitable for any intended use or that these programs
   will work without errors in any combination with the data processing environment. Providing
   you with these software programs shall neither constitute a claim for technical support nor
   for any other remedy for defects. Any claims for damages of any nature and for any legal
   reason arising from installing or using these software programs or program modules are ex-
   cluded, unless these damages was caused by Bosch Rexroth`s statutory representatives or em-
   ployees by wilful misconduct or by gross negligence or liability is compulsory in accordance
   with the German product liability law. In any case Bosch Rexroth`s liability for any conse-
   quential or incidental damages such as, but not limited to loss of profit, loss of pro-
   duction or loss of data is excluded.      
*)
(*---------------------------------------------------------------------------------------------*)

VAR_INPUT
	// Internal references to the extension
    // this references include the base and the extensions, the refererences without Ext include only the base 
    (* arAxisCtrl_gb *)
    AdminCtrlExt     : REFERENCE TO TE_AXIS_ADMINISTRATION; (* Administration of the axis *)
    PosModeCtrlExt   : REFERENCE TO TE_AXIS_POSITIONING;    (* Operating mode absolute positioning *)
    VelModeCtrlExt   : REFERENCE TO TE_AXIS_VELOCITY;       (* Operating mode velocity control *)
    SyncModeCtrlExt  : REFERENCE TO TE_AXIS_SYNCHRONISATION;(* Operating mode synchronisation (phs,vel,and cam)*)
    (* arAxisStatus_gb *)
    AdminStatusExt   : REFERENCE TO TE_AXIS_ADMIN_STATUS;   (* Status administration of the axis *)
    DiagStatusExt    : REFERENCE TO TE_AXIS_DIAGNOSIS;      (* Axis diagnosis information, error, warning.... *)
    PosStatusExt     : REFERENCE TO TE_AXIS_POS_STATUS;     (* Status operating mode positioning *)
    VelStatusExt     : REFERENCE TO TE_AXIS_VEL_STATUS;     (* Status operating mode velocity control *)
    SyncModeStatusExt: REFERENCE TO TE_AXIS_SYNC_STATUS;    (* Status op mode synchronisation (phs,vel,and cam)*)
    // add user extensions below here
    SetupMode: REFERENCE TO TE_AXIS_SETUP_MODE; 
    SetupModeAck: REFERENCE TO TE_AXIS_SETUP_MODE_STATUS; 
	AxisData_HMI: REFERENCE TO TE_AXIS_DATA_STATUS;
END_VAR
VAR_OUTPUT

END_VAR
VAR
  udiCycleCntInP4: UDINT; // count cycles in P4 to spread the parameter write load
  //######  SetupMode ######## 
  bLatchSetupModeEnable:  BOOL;
  enOriAxisMode:  MB_AXIS_MODE; 	// stored OpMode, when SetupMode is activated. reset when SetupMode is left
  enMyActAxisMode:  MB_AXIS_MODE;	// actual Setup-OpMode, used to detect when the OpMode is changed during active SetupMode  
  uiHomingState: UINT;
  // define as RETAIN (global) when arAxisCtrl_gb is RETAIN 
  bOriValuesStored:  BOOL;
  rOriVel:  REAL;
  rOriAccel:  REAL;
  rOriDecel:  REAL;
  rOriPos:    REAL;
  rOriVelPos: REAL;
  rOriAccelPos: REAL;
  rOriDecelPos: REAL;
  //######  Homing ########
  bHomingOld: BOOL:=FALSE;  // to detect the falling edge
  bHomingRemovedBeforeFinished: BOOL:= FALSE;
  bAbsoluteEncoder: BOOL:=FALSE;
  diParameterS277: DINT:=0;
  MB_ReadParameterS277: MB_ReadParameter;

  //######  AngleOffset ######## 
  // Remember AngleOffset to write only on changes 
  rLastAngleOffset:  REAL := 0.01; // default old value not equal 0 to enforce a transmission 
  // Write AngleOffset 
  fbWrAngleOffs:       MB_WriteRealParameter;
  bExecWrAngleOffs:    BOOL:=FALSE;

  //######  SyncAcceleration ######## 
  // Remember SyncAcceleration to write only on changes 
  rLastSyncAcc:      REAL := 0.01; // default old value not equal 0 to enforce a transmission 
  // Write SyncAcceleration 
  fbWrSyncAcc:       MB_WriteRealParameter;
  bExecWrSyncAcc:    BOOL:=FALSE;

  //######  Syncvelocity ######## 
  // Remember Syncvelocity to write only on changes 
  rLastSyncVel:      REAL := 0.01; // default old value not equal 0 to enforce a transmission 
  // Write SyncAcceleration 
  fbWrSyncVel:       MB_WriteRealParameter;
  bExecWrSyncVel:    BOOL:=FALSE;
  
  //######  PhasingMaster ######## 
  fbAxisPhasing: MB_Phasing;
  bExecPhasing:    BOOL:=FALSE;
  rOldPhaseShift: REAL := 0.01;  // default old value not equal 0 to enforce a transmission 
  bInitFirst: BOOL := FALSE;
  
  //######  RetriggerOpMode ######## 
  bRetriggerOpModeOld: BOOL;
  bOriginalOpMode: MB_AXIS_MODE;
  bOpModeChanged: BOOL;
	
	//######  Activate PM for special axis errors ########
  bOriginalPM: BOOL;
	uiStatePM: UINT :=STATE_ERR_IDLE;
  
END_VAR
VAR CONSTANT  
  MASK_MODE_ANGLE_OFFSET    :WORD := 16#0B00; // SYNC_CAM, SYNC_PROFILE, FLEX_PROFILE 
  
  STATE_HOMING_START         :UINT := 0;
  STATE_HOMING_READ_S277     :UINT := 1;
  STATE_HOMING_ABS_REAL_AXIS :UINT := 2;
  STATE_HOMING_INC_REAL_AXIS :UINT := 3;
  STATE_HOMING_VIRT_AXIS     :UINT := 5;
  STATE_HOMING_FINISHED      :UINT := 6;
  STATE_HOMING_NOT_POSSIBLE  :UINT := 9;
  STATE_HOMING_ERROR         :UINT := 10;

  // States of special error handling  
	STATE_ERR_IDLE             :UINT := 0;
	STATE_ERR_ACTIVATE_PM      :UINT := 1;
	STATE_ERR_ACTIVATE_OM      :UINT := 2;

  // state machine error
  HOMING_STATE_MACHINE_ERR: ERROR_STRUCT := ( Table := USER10_TABLE, Additional1 := 16#00004201, Additional2 := 16#00000000);
  // Homing not implemented for control axis
  HOMING_CONFIGURATION_ERR: ERROR_STRUCT := ( Table := USER10_TABLE, Additional1 := 16#00004202, Additional2 := 16#00000000);
  // SetupMode is only allowed when in Modeab or ModeAH
  SETUPMODE_OPMODE_ERR: ERROR_STRUCT := ( Table := USER10_TABLE, Additional1 := 16#00004203, Additional2 := 16#00000000);
END_VAR

// Handle RetriggerOpMode 
// Do this before calling the base FB to be able to overwrite the OpMode set cyclic by the user.
actRetriggerOpMode();
// Activate PM for special axis errors. In case of drive error F8022 and F8042 switch to PM to clear this error.
// Do this before calling the base FB to be able to overwrite the paramLevel set cyclic by the user.
// Defdb00147736: uncomment the next line to activate the special error handling.  
// actPMSpecialErrors(); 

(* call the base FB, call it first, to have the information AdminStatus.Active actual *)
SUPER^();

(* 2nd check, if the axis is active *)
IF AdminStatus.Active = FALSE THEN	
  RETURN;
END_IF;
// Check if we are in bb. A-0-0021 is read internal by the MB_AxisInterfaceType01
// Bit 12 of A-0-0021 means "Axis is in operation mode (P4)" 
// When all axes in parallel write parameters, we overload the system. So we
// count the cycles and distribute the load with using the axis address  
IF AxisData[AdminCtrl.Axis.AxisNo].Axis_OperationMode = TRUE THEN 
  udiCycleCntInP4 := udiCycleCntInP4 + 1;
ELSE
  udiCycleCntInP4 := 0;
END_IF

(* add your extensions below here, keep the elements above
   Erweiterungen hier einfuegen, Elemente oberhalb nicht veraendern *)
(* user extensions | Anwender Erweiterungen *)

(* Jog/Home an axis within the AxisInterface *)
actSetupMode();

(* Write the Angle offset begin of profile A-0-2730 *)
actAngleOffset();

(* Write the Sync Acceleration into A-0-2791 *)
(* and the Sync Velocity into A-0-2790 *)
actSyncAccVel();

(* Handle PhasingMaster *)
actPhaseShift();

(* copy AxisData status informations to AxisData_HMI structure to transmit to HMI *)
actCopyAxisData_HMI();

ACTION actRetriggerOpMode:
// Restart the same OpMode again, e.g. MoveRelative with same distance
// Detect rising edge on input RetriggerOpMode
IF AdminCtrlExt.RetriggerOpMode AND NOT bRetriggerOpModeOld THEN
  // set ModeExternalFb for one cycle
    bOriginalOpMode := AdminCtrlExt._OpMode.en ;
    AdminCtrlExt._OpMode.en := ModeExternalFb;
    bOpModeChanged :=TRUE;
ELSIF bOpModeChanged THEN
    // reset OpMode to original in next cycle
    AdminCtrl._OpMode.en := bOriginalOpMode;
    bOpModeChanged :=FALSE; 
END_IF
bRetriggerOpModeOld  := AdminCtrlExt.RetriggerOpMode;
END_ACTION

ACTION actPMSpecialErrors:
// Activate PM of the axis if special drive errors occur 

{IF defined(variable: AdminCtrl.ParamLevel)}
CASE uiStatePM OF
  
STATE_ERR_IDLE: 
  // ---------------------------------------------------------
  // Idle state --> do nothing
	// ---------------------------------------------------------
  // Wait until F8022 or F8042 error occurs   
	IF (DiagStatus.Number = 16#F2008022) OR (DiagStatus.Number = 16#F2008042) THEN
		bOriginalPM := AdminCtrl.ParamLevel;
    uiStatePM := STATE_ERR_ACTIVATE_PM;	
	END_IF
	
STATE_ERR_ACTIVATE_PM:
  // ---------------------------------------------------------
  // Command axis to Parameter mode "PM"  
	// ---------------------------------------------------------
  AdminCtrl.ParamLevel := TRUE;
 
	// Wait until error disappears
	IF (DiagStatusExt.Error = FALSE ) THEN
    uiStatePM := STATE_ERR_ACTIVATE_OM;	
	END_IF
 
STATE_ERR_ACTIVATE_OM: 
  // ---------------------------------------------------------
  // Command axis to Operation Mode "OM" 
  // --------------------------------------------------------- 
  AdminCtrl.ParamLevel := FALSE;
 
  // Wait untill axis is in OM 
  IF AxisData[AdminCtrl.Axis.AxisNo].Axis_OperationMode = TRUE THEN
    uiStatePM := STATE_ERR_IDLE;	
		AdminCtrl.ParamLevel := bOriginalPM;
	END_IF

END_CASE
{END_IF}
;
END_ACTION

METHOD mClearError : BOOL
VAR_INPUT
	boClearError : BOOL;
END_VAR
VAR
END_VAR
IF ADR(AdminCtrlExt) <> 0 THEN // check if the references are set (not needed, when references are set in FB_Init)
  AdminCtrlExt.ClearError := boClearError;
END_IF
IF ADR(DiagStatusExt) <> 0 THEN // check if the references are set (not needed, when references are set in FB_Init)
  mClearError := DiagStatusExt.Error;
END_IF
END_METHOD

ACTION actPhaseShift:
//***************************************************************
// Implements a PhasingMaster with the function block MB_Phasing
//***************************************************************
//********* handle phase offset when sync-mode is active *******
IF( ((INT_TO_WORD(AdminStatusExt._OpModeAck) AND MASK_MODE_PHASE_OFFSET) <> 0) )THEN
  IF( rOldPhaseShift <> SyncModeCtrlExt.PhaseShift) THEN
    // start transmission 
	SyncModeStatusExt.PhasingMasterDone := FALSE;
	bExecPhasing := TRUE;
  END_IF
  IF fbAxisPhasing.Done THEN
    // finished GOOD transmission 
	SyncModeStatusExt.PhasingMasterDone := TRUE;
	bExecPhasing := FALSE;
    // remember old value 
    rOldPhaseShift := SyncModeCtrlExt.PhaseShift;
  ELSIF (fbAxisPhasing.Error = TRUE) THEN
    // finished BAD transmission 
	bExecPhasing := FALSE;
    SUPER^.mSetError( Error      := TRUE, 
                      ErrorID    := fbAxisPhasing.ErrorID, 
                      ErrorIdent := fbAxisPhasing.ErrorIdent);
  END_IF
  // keep the FB always active to generate PhasingMasterDone 
  fbAxisPhasing(
    Execute      := bExecPhasing,
    PhaseShift   := SyncModeCtrlExt.PhaseShift,
    Velocity     := SyncModeCtrlExt.PhaseShiftVel,
    Acceleration := SyncModeCtrlExt.PhaseShiftAcc,
    Axis         := AdminCtrlExt.Axis );
ELSE
  SyncModeStatusExt.PhasingMasterDone := FALSE; // Reset, when no Sync-Mode active 
END_IF // end of 'IF( (INT_TO_WORD(AdminStatusExt._OpMode.enAck) AND MASK_MODE_PHASE_OFFSET) <> 0 ) THEN'
END_ACTION

ACTION actAngleOffset:
// Implements writing the angle offset into parameter A-0-2730
// Check if we are in bb. Otherwise we get errors.
// Do this only when sync is supported and the parameters are available.
// Distribute the load with using the axis address
IF AxisData[AdminCtrlExt.Axis.AxisNo].Axis_OperationMode = TRUE   AND
   AdminStatusExt.AxisFeatures.OPMODE_SYNC = TRUE                 AND 
   (udiCycleCntInP4 > DINT_TO_UDINT(2 * AdminCtrlExt.Axis.AxisNo))    THEN 
  // write angle offset when changed 
  IF SyncModeCtrlExt.AngleOffset <> rLastAngleOffset THEN
    // start transmission 
    SyncModeStatusExt.AngleOffsetDone := FALSE;
    bExecWrAngleOffs := TRUE;
  END_IF
  IF fbWrAngleOffs.Done = TRUE THEN 
    // finished GOOD transmission 
    SyncModeStatusExt.AngleOffsetDone := TRUE;
    bExecWrAngleOffs := FALSE;
    // remember old value 
    rLastAngleOffset := SyncModeCtrlExt.AngleOffset;
  ELSIF fbWrAngleOffs.Error = TRUE THEN  
    // finished BAD transmission 
    bExecWrAngleOffs := FALSE;
    SUPER^.mSetError( Error      := TRUE, 
                      ErrorID    := fbWrAngleOffs.ErrorID, 
                      ErrorIdent := fbWrAngleOffs.ErrorIdent);
  END_IF  
  // call write parameter FB 
  fbWrAngleOffs(
	Execute:= bExecWrAngleOffs, 
	ParameterNumber:= FP_A_0_2730, 
	Value:= SyncModeCtrlExt.AngleOffset, 
	Axis:= AdminCtrlExt.Axis );	
ELSE
  // reset FBs when not in bb 
  fbWrAngleOffs( Execute:= FALSE, Axis:= AdminCtrlExt.Axis );	
END_IF	
// to avoid service channel transmissions (interpolation drive), place the P-0-0061 into 
// an MDT data container (here e.g. container A) and write to the data container
//AxisData[AdminCtrlExt.Axis].dwUserCmdDataA_q.REAL_ := SyncModeCtrlExt.AngleOffset;
END_ACTION

METHOD mGetOpMode : MB_AXIS_MODE
VAR_INPUT
END_VAR
VAR
END_VAR
IF ADR(AdminStatusExt) <> 0 THEN // check if the references are set (not needed, when references are set in FB_Init)
  mGetOpMode := AdminStatusExt._OpModeAck;
END_IF
END_METHOD

METHOD mSetOpMode : MB_AXIS_MODE
VAR_INPUT
	enOpMode: MB_AXIS_MODE;
END_VAR
VAR
END_VAR
IF ADR(AdminCtrlExt) <> 0 THEN // check if the references are set (not needed, when references are set in FB_Init)
  AdminCtrlExt._OpMode.en := enOpMode;
END_IF
IF ADR(AdminStatusExt) <> 0 THEN // check if the references are set (not needed, when references are set in FB_Init)
  mSetOpMode := AdminStatusExt._OpModeAck;
END_IF
END_METHOD

